FUNCTION_BLOCK FB_LidFeeder
VAR_INPUT
	_CONTROL_:BOOL;	
	bEnable:BOOL;						//Zezowlenie na pracę podajnika platynek
	bEStop:BOOL;						//Stop awaryjny nieaktywny
	bHeaterEnable:BOOL; 				//Zezwolenie na pracę grzałki wstępnej
	bRunPrepare:BOOL;							//Zezwolenie na podanie platynki. Podajnik platynek podczas cyklu podawania musi mieć załączony ten bit. Po wykonaniu podawania (kiedy status podajnika jest "LidPutted"), bit powinien być wyłączony. Dopiero kolejne załączenie pozwoli na podanie platynki
	bRun: BOOL;						//Zezwolenie na ostatni ruch opuszczania platynki
	bHoming:BOOL;						//Zezwolenie na wykonanie bazowania i pozycjonowania podajnika
	bHeightSet:BOOL;					//Ustaw wysokość
	bIgnoreError:BOOL;					//Ignorowania błędów cyklu pracy
	bReset:BOOL;						//Reset błędu, jeśli w stanie "eError"
	nLidHeatingTime:INT;				//Czas zgrzewania wstępnego [ms]
	nPositionHeightSV:LREAL;			//Wysokość zadana na której ma znajdować się podajnik
	bHeaterTemperatureErrorIgnore:BOOL; //Zmienna pozwalająca ignorowanie aktualnej temperatury
	bManualMovement:BOOL; 			//Uruchomienie trybu ruchów ręcznych
	HEATER_PARAMETERS_:BOOL;	
	nHeaterTemperatureSV:INT;			//Zadana wartość grzałki podajnika platynek
	rKp:REAL;							//Wzmocnienie proporcjonalne regulatora grzałki
	rTd:REAL;							//Czas różniczkowania regulatora grzałki
	rTi:REAL;							//Czas całkowania regulatora grzałki
	//nCycle:INT;						//Czas okresu PWM grzałki [s]
	nTempHisteresis:INT;				//Dopuszczalna różnica pomiędzy wartością zadaną a aktualną [st. C]				
	lrMaxHeight:LREAL;					//Maksymalna wysokość podajnika platynek
	lrMinHeight:LREAL;					//Minimalna wysokość podajnika platynek

	_SENSORS_:BOOL;
	bFeederActuatorUpSensor1:BOOL;		//krańcówka górna podajnika platynek
	bFeederActuatorDownSensor1:BOOL;	//krańcówka dolna podajnika platynek
	bFeederActuatorDownSensor2:BOOL;	//krańcówka dolna podajnika platynek
	bLidSuckedSensor:BOOL;				//Czujnik zassania platynki, zassana jesli TRUE
	lrHeaterTemperatureCVSensor:LREAL;	//Wartość aktualna temperatury grzałki
	bTemperatureSensorFault:BOOL;		//Błąd czujnika temperatury
	nPositionHeightCV:LREAL;			//Aktualna wysokość podajnika platynek

	_HEIGHTMOTOR_ :BOOL;	
	bHeightMotorEncoderPulse :BOOL;			//Sygnał impulsów enkodera siłownika
	rHeightMotorPositionOffset :REAL;		//Wysokość bazowani podnośnika

	_ALARMINFO_ :BOOL;
	iStationIndex:UDINT;					//Numer stacji 
	sStationName:STRING;					//Nazwa stacji	

	bLidFeederLowLevelSensor			: BOOL;		// Czujnik niskiego poziomu platynek w zasobniku
	bEmergencyUp						: BOOL;		
	//Vasyl 24.10.25 aktualizacja bloczka enkodera
	udiHeightMotorEncoderCV		: UDINT;
	bHeightEncoderSetCDone		: BOOL;	
	
END_VAR
VAR_OUTPUT
	bHeaterPWMOut :BOOL;					//Wyjscie PWM sterujące grzałką
	eState: E_Station;						//Stan ogólny bloku
	eRunningState: E_LidFeederState;		//Stan podajnika platynek
	bError: BOOL;							//Błąd stacji
	nErrorNr: UDINT;						//Nr błędu podajnika platynek
	sErrorDescription:STRING(200);			//Opis błędu
	sErrorDescription2: STRING(200);		//Opis błędu 2
	sErrorStationName:STRING;				//Nazwa stacji
	udiStationID:UDINT;						// Nr stacji

	bLidFeederActuator1:BOOL;				//Sterownie siłownika podajnika platynek
	bLidFeederActuator2:BOOL;				//Sterownie siłownika podajnika platynek
	bLidHeaterActuator:BOOL;				//Sterowanie siłownika grzałki wstępnej
	bLidSuckerActuator:BOOL;				//Sterowanie zasysaniem platynek
	bHeightMotorUp:BOOL;					//Sterowanie silnikiem podnośnika  - RUCH W GÓRĘ
	bHeightMotorDown:BOOL;					//Sterowanie silnikiem podnośnika  - RUCH W DÓŁ
	lrHeightMotorCV:LREAL;					//Aktualna pozycja podnośnika
	tCycleTime:TIME;	
	bHomingDone:BOOL;						//Wymagane ponowne bazowanie (blad podczas bazowania lub stop awaryjny)	
	bCycleDone:BOOL;
	bCycleNotDone:BOOL;
	//Vasyl 24.10.25 aktualizacja bloczka enkodera
	udiHeightMotorEncoderSetCV	: UDINT;		
	bHeightEncoderSetC			: BOOL;					// Zerowanie enkodera
	
END_VAR
VAR
	nSuckingRetry: INT;						//Licznik nieudanego pobrania platynki
	tonHeatingTime: TON;					//Timer czasu zgrzewania platynki
	tonLidSuckingDelay: TON; 				//Timer opóźnienia zassania po włączeniu eżektora w stanie zasysania
	tonHeightNoChange: TON; 				//Timer wykrycia braku ruchu siłownika zmiany wysokości stacji
	nLastPositionHeightCV: LREAL;			//Pozycja podnośnika w poprzednim cyklu programu
	tonErrorHeightChange: TON; 				//Timer błędu podnośnika

	rtEncoderHomed:R_TRIG;
	tonCycleTimer:TON;
	rtrigCycleTimerRead:R_TRIG;
	
	tonLimitPosMinReachedDelay: TON;
	tonLimitPosMaxReachedDelay: TON;
	tonMaxHeight: TON;
	tonLidFeederActuator1DownError: TON;
	tonLidFeederActuator1UpError: TON;
	tonLidFeederActuator2DownError: TON;
	//Podnośnik Jiesang	
	fbHeightMotorEncoder: FB_JiesangActuatorEncoderModul;	// Blok enkodera podnośnika chwytaka stabilizującego pod zakręcarką	
	bHeightMotorEncoderCounterReset:BOOL; 				//Sygnał resetu enkodera
	bHeightMotorEncoderHomed:BOOL;						//Informacja od enkodera że jest zbazowany

	eLastState: E_Station;							//Stan ogólny bloku
	eLastRunningState: E_LidFeederState;			//Stan podbloku
	eLastStateTemp: E_Station;						//Stan ogólny bloku
	eLastRunningStateTemp: E_LidFeederState;		//Stan podbloku
	bStateError: BOOL;
	tonEstopDelay: TON;
	
	fbTempRegulator				: FB_TempRegulator;
	bTempRegulatorReset			: BOOL;
	
	tofbHeaterPWMOut					: TOF;
	tonHeaterOnAndNotHeating			: TON;
	lrHeaterTemperatureCVSensorLast		: LREAL;	//Wartość aktualna temperatury grzałki
	tonHeaterOnAndSensorShows0			: TON;
	tofHeightMotorDown: TOF;
	tonbLidFeederLowLevelSensor: TON;
	ftWarning: F_TRIG;
	tonbLidFeederWellLevel: TON;
	rtbHeightMotorEncoderPulse: R_TRIG;
	ftbHeightMotorEncoderPulse: F_TRIG;
	lrHeightMotorEncoderPulses: LREAL;

	bLidFeederActuator1LastState		: BOOL;	//Stan przed Manual
	bLidFeederActuator2LastState		: BOOL;	//Stan przed Manual
	bLidSuckerActuatorLastState			: BOOL;	//Stan przed Manual
	bLidHeaterActuatorLastState			: BOOL;	//Stan przed Manual
	tonGoingUp: TON;
	
	//Zmienne od EVENTLOGGER
	bAlarmInit 						: BOOL := TRUE; 
	nAlarmNumerator					: INT;
	arfbAlarm						: ARRAY[0..19] OF  FB_TcAlarm;		//Tablica bloczków błędów
	fbSourceInfo 					: FB_TcSourceInfo;
	iSourceInfo						: I_TcSourceInfo;
	sAlarmTest						: STRING;
	//Koniec zmiennych od EVENTLOGGER
END_VAR

VAR_IN_OUT
	bManualLidFeederActuator1:BOOL;		//Ruch ręczny siłownikiem podajnika platynek
	bManualLidFeederActuator2:BOOL;		//Ruch ręczny siłownikiem 2 podajnika platynek
	bManualLidSuckerActuator:BOOL;		//Ręczne załączenie zassania platynek
	bManualLidHeaterActuator:BOOL;		//Ruch ręczny siłownika grzałek;
	bManualHeightMotorUp:BOOL;			//Ruch ręczny podnośnika stacji w górę
	bManualHeightMotorDown:BOOL;		//Ruch ręczny podnośnika stacji w dół
	
	bWarning							: BOOL;
END_VAR

Signals();
HeightMotor();
ErrorHandling();
Control();
HeaterRegulator();
Statistics();
EncoderTest();
aStationID();
(*Zapisywanie ostatniego stanu*)
IF eLastStateTemp<>eState THEN
	eLastState := eLastStateTemp;
END_IF
eLastStateTemp := eState;
IF eLastRunningStateTemp<>eRunningState THEN
	eLastRunningState := eLastRunningStateTemp;
END_IF
eLastRunningStateTemp := eRunningState;
(*Koniec Zapisywanie ostatniego stanu*)

nLastPositionHeightCV:=nPositionHeightCV;

ACTION aStationID:
udiStationID	:=	iStationIndex;
END_ACTION

ACTION Control:

	(** TIMERY**)
	rtEncoderHomed(CLK:=bHeightMotorEncoderHomed,Q=>);
	tonHeightNoChange(IN:=((bHeightMotorUp OR bHeightMotorDown) AND nLastPositionHeightCV=nPositionHeightCV), PT:=T#1S); 
	tonLimitPosMinReachedDelay(IN:=(nPositionHeightCV<=lrMinHeight) AND eState=E_Station.eHoming,PT:=T#2S);
	tonLimitPosMaxReachedDelay(IN:=(nPositionHeightCV>=lrMaxHeight) AND eState=E_Station.eHoming,PT:=T#2S);

	(*****Wyłączenie enable*****)
	IF NOT bEnable THEN
		IF eState <> E_Station.eDisabled AND eState <> E_Station.ePreparingToDisable THEN
				eState 				:= E_Station.ePreparingToDisable; 
		END_IF	
	END_IF

	(*****Estop*****)
	IF NOT bEstop  THEN	
		IF eState <> E_Station.eAborted AND eState <> E_Station.eAborting AND eState <> E_Station.eDisabled THEN
				eState 				:= E_Station.eAborting; 
		END_IF
	END_IF
	
	IF bEstop AND bEmergencyUp THEN
		eState 				:= E_Station.eAborting;
	END_IF

	
	CASE eState OF
	/////////////////////////////	
		E_Station.eDisabled: 					// Stan nieaktywnosci (Stacja wyłączona) 
		
			IF bEnable THEN
				eState 				:= E_Station.ePreparingToReady; 
			END_IF 
			
    /////////////////////////////	    
		E_Station.eAborted: 					// Stan bezpiecznego zatrzymania (po Abortingu) 

			IF bEStop THEN
				eState 				:= E_Station.ePreparingToReady;
			END_IF
			
	/////////////////////////////	
		E_Station.eAborting:                 	// Stan bezpiecznego zatrzymywania (po EStopie)
		
			IF NOT bEstop THEN
				
				bLidFeederActuator1		:=	FALSE;
				bLidFeederActuator2		:=	FALSE;
				bLidSuckerActuator		:=	FALSE;
				bLidHeaterActuator		:=	FALSE;
				bHeightMotorDown		:=	FALSE;
				bHeightMotorUp			:=	FALSE;	
				eState 					:=	E_Station.eAborted;  
				eRunningState			:=	E_LidFeederState.eDisabled;
				
			ELSIF bEmergencyUp THEN
			
				bHeightMotorUp			:= NOT tofHeightMotorDown.Q;
				bHeightMotorDown		:= FALSE;
				bLidFeederActuator1		:= FALSE;
				bLidFeederActuator2		:= FALSE;
				bLidSuckerActuator		:= FALSE;	
				bHeightMotorDown		:= FALSE;
				
				bHomingDone 			:= FALSE;
				
				IF tonHeightNoChange.Q THEN
					bHeightMotorEncoderCounterReset	:= TRUE;
					bHeightMotorUp					:= FALSE;
				END_IF
				
				
			END_IF
	/////////////////////////////			
		E_Station.eError:                 	 	// Stan błędu 	
		
					bLidFeederActuator1	:=FALSE;
		            bLidFeederActuator2	:=FALSE;
					bLidSuckerActuator	:=FALSE;
	
			IF bReset THEN
				eState 				:= E_Station.eResetting;
			END_IF
			
	/////////////////////////////
		E_Station.eResetting:					// Stan resetowania bledu (po Errorze)

		
// 			CASE nErrorNr-iStationIndex OF
// 		
// 				//Error 1 - ZBYT DLUGIE ZASYSANIE
// 				221:
// 					bError := FALSE;
// 				ELSE
// 					bError := FALSE;	
// 		END_CASE
			// 			
			bLidFeederActuator1	:=FALSE;
            bLidFeederActuator2	:=FALSE;
			bLidSuckerActuator	:=FALSE;
			
			IF NOT bError THEN
				nErrorNr 			:=	0;
   				sErrorDescription 	:=	'';
				bTempRegulatorReset	:=	FALSE;
				eState 				:=	E_Station.ePreparingToReady;
			ELSE
				eState 				:=	E_Station.eError;
			END_IF
        
	/////////////////////////////
		E_Station.eManualMovement:     			// Stan ruchów manualnych  
       
			ManualMovements();
			//Wyjście z trybu serwisowego
			IF NOT bManualMovement THEN
				bLidFeederActuator1		:=	bLidFeederActuator1LastState ;//:=FALSE;
				bLidFeederActuator2		:=	bLidFeederActuator2LastState ; //:=FALSE;
				bLidSuckerActuator		:=	bLidSuckerActuatorLastState ;//:=FALSE;
				bLidHeaterActuator		:=	bLidHeaterActuatorLastState ;//:=FALSE;
				bHeightMotorDown		:=	FALSE;
				bHeightMotorUp			:=	FALSE;
				eState:=E_Station.eReady;
			END_IF

	/////////////////////////////
		E_Station.eHoming:						// Stan bazowania 

			Homing();
			IF NOT bHoming AND NOT bHeightSet THEN
			   eState:=E_Station.ePreparingToReady;
			   	bHeightMotorDown:=FALSE;
				bHeightMotorUp:=FALSE;
			END_IF		
			
	/////////////////////////////
		E_Station.eHomingDone:                  // Stan wykonania bazowania 
		
			bHeightMotorDown:=FALSE;
			bHeightMotorUp:=FALSE;
			bHeightMotorEncoderCounterReset:=FALSE;
			bHomingDone:=TRUE;
			IF NOT bHoming AND NOT bHeightSet THEN
			  	 eState:=E_Station.eReady;
			END_IF
			
	/////////////////////////////
		E_Station.ePreparingToReady:            // Stan przygotowywania do gotowosci (zawsze przed Ready)  
		
			bLidFeederActuator1		:=	FALSE;
			bLidFeederActuator2		:=	FALSE;
			//bLidSuckerActuator		:=	FALSE; //Zmiana LU205
			bLidHeaterActuator		:=	FALSE;
			eRunningState:=E_LidFeederState.eReady;
			eState:=E_Station.eReady;	
			
	/////////////////////////////
		E_Station.ePreparingToDisable:          // Stan przygotowywania do nieaktywnosci (po wyłączeniu Enable) 
  
			bLidFeederActuator1		:=	FALSE;
			bLidFeederActuator2		:=	FALSE;
			bLidSuckerActuator		:=	FALSE;
			bLidHeaterActuator		:=	FALSE;
			
			bHeightMotorUp:=TRUE;
			bHeightMotorDown:=FALSE;	
			IF tonHeightNoChange.Q THEN
				bHeightMotorUp:=FALSE;
				bHeightMotorDown:=FALSE;	
				eState:=E_Station.eDisabled;
				eRunningState:=E_LidFeederState.eDisabled;
			END_IF
			
			
	/////////////////////////////
		E_Station.eReady:						// Stan gotowosci 
		
			IF bRunPrepare OR bRun AND (NOT bCycleDone AND NOT bCycleNotDone) THEN
				eState 				:= E_Station.eStarting; 
			END_IF
			IF bHoming OR bHeightSet THEN
				eState 				:= E_Station.eHoming; 
			END_IF
			IF bManualMovement THEN
				//Jeśli przejście w tryb ruchów manualnych przepisz wszystkie stany siłowników sterowanych przez moduł
				//aby zapobiec ewentualnym kolizjom po wejściu w tryb serwisowy
				bManualLidFeederActuator1	:= bLidFeederActuator1LastState :=	bLidFeederActuator1;
				bManualLidFeederActuator2	:= bLidFeederActuator2LastState :=	bLidFeederActuator2;
				bManualLidSuckerActuator	:= bLidSuckerActuatorLastState 	:=  bLidSuckerActuator;
				bManualLidHeaterActuator	:= bLidHeaterActuatorLastState	:=	bLidHeaterActuator;
				bManualHeightMotorUp		:=	bHeightMotorUp;
				bManualHeightMotorDown		:=	bHeightMotorDown;
				
				eState 						:=	E_Station.eManualMovement; 
			END_IF
			IF NOT bRun THEN
				bCycleDone 					:= FALSE;
				bCycleNotDone 				:= FALSE;			
			END_IF
			
	/////////////////////////////
		E_Station.eStopping:					// Stan zatrzymywania 
		
			Running();
			IF eRunningState=E_LidFeederState.eReady THEN
				eState 	:= E_Station.eReady;
			END_IF
			//eState 					:= E_Station.eReady;	
			
	/////////////////////////////
		E_Station.eStarting:                  	// Stan uruchamiania (po Ready)
		
			eState					 := E_Station.eRunning; 
			
	/////////////////////////////
		E_Station.eRunning:              		// Stan wykonywania cyklu (po Startingu), w tym stanie osobny
 
			Running();
			IF NOT bRunPrepare THEN					(*Przerywanie cyklu*)
				eState 				 := E_Station.eStopping;	
			END_IF
			IF bCycleDone OR bCycleNotDone THEN (*Cykl zakończony*)
				eState 				 := E_Station.eReady;
			END_IF	
	/////////////////////////////		
	END_CASE
END_ACTION

ACTION EncoderTest:


rtbHeightMotorEncoderPulse(CLK:=bHeightMotorEncoderPulse,Q=>);
ftbHeightMotorEncoderPulse(CLK:=bHeightMotorEncoderPulse,Q=>);


IF rtbHeightMotorEncoderPulse.Q THEN
	lrHeightMotorEncoderPulses	:=	lrHeightMotorEncoderPulses +	1;
END_IF
END_ACTION

ACTION ErrorHandling:
// Alarm_0340	340	Error	Zbyt długa próba zassania platynki - uzupełnij platynki lub popraw ich położenie
// Alarm_0341	341	Error	Nieudana próba podania platynki - zwiększ ciśnienie
// Alarm_0342	342	Error	Błąd czujnika temperatury grzałki - sprawdź połączenie
// Alarm_0343	343	Error	Blokada podnośnika lub brak zasilania - sprawdź czujnik lub odblokuj mechanicznie
// Alarm_0344	344	Error	Wartość zadana wysokości jest większa od maksymalnej - zmień ustawienia w recepturze
// Alarm_0345	345	Error	Blokada siłownika dolnego podczas opuszczania - sprawdź czujnik
// Alarm_0346	346	Error	Blokada siłownika dolnego podczas podnoszenia - sprawdź czujnik
// Alarm_0347	347	Error	Blokada siłownika górnego podczas opuszczania - sprawdź czujnik
// Alarm_0348	348	Error	Błąd grzania, brak wzrostu temperatury - sprawdź czujnik
// Alarm_0349	349	Error	Błąd grzania, brak sygnału z czujnika temperatury - sprawdź czujnik

IF bAlarmInit THEN
    bAlarmInit := FALSE; 
	fbSourceInfo.Clear();
	fbSourceInfo.sName:=sStationName;//'Machine';
	fbSourceInfo.nId:=udiStationID;//2700;
	// Alarm_0340	340	Error	Zbyt długa próba zassania platynki - uzupełnij platynki lub popraw ich położenie
    arfbAlarm[0].CreateEx(stEventEntry := TC_EVENTS.AlarmClass.Alarm_0340, bWithConfirmation:= FALSE,  ipSourceInfo:= fbSourceInfo); 
	// Alarm_0341	341	Error	Nieudana próba podania platynki - zwiększ ciśnienie
	arfbAlarm[1].CreateEx(stEventEntry := TC_EVENTS.AlarmClass.Alarm_0341, bWithConfirmation:= FALSE,  ipSourceInfo:= fbSourceInfo); 
	//// Alarm_0342	342	Error	Błąd czujnika temperatury grzałki - sprawdź połączenie
	//arfbAlarm[2].CreateEx(stEventEntry := TC_EVENTS.AlarmClass.Alarm_0342, bWithConfirmation:= FALSE,  ipSourceInfo:= fbSourceInfo); 
	// Alarm_0343	343	Error	Blokada podnośnika lub brak zasilania - sprawdź czujnik lub odblokuj mechanicznie
	arfbAlarm[3].CreateEx(stEventEntry := TC_EVENTS.AlarmClass.Alarm_0343, bWithConfirmation:= FALSE,  ipSourceInfo:= fbSourceInfo); 
	// Alarm_0344	344	Error	Wartość zadana wysokości jest większa od maksymalnej - zmień ustawienia w recepturze
	arfbAlarm[4].CreateEx(stEventEntry := TC_EVENTS.AlarmClass.Alarm_0344, bWithConfirmation:= FALSE,  ipSourceInfo:= fbSourceInfo); 
	// Alarm_0345	345	Error	Blokada siłownika dolnego podczas opuszczania - sprawdź czujnik
	arfbAlarm[5].CreateEx(stEventEntry := TC_EVENTS.AlarmClass.Alarm_0345, bWithConfirmation:= FALSE,  ipSourceInfo:= fbSourceInfo); 
	// Alarm_0346	346	Error	Blokada siłownika dolnego podczas podnoszenia - sprawdź czujnik
	arfbAlarm[6].CreateEx(stEventEntry := TC_EVENTS.AlarmClass.Alarm_0346, bWithConfirmation:= FALSE,  ipSourceInfo:= fbSourceInfo); 
	// Alarm_0347	347	Error	Blokada siłownika górnego podczas opuszczania - sprawdź czujnik
	arfbAlarm[7].CreateEx(stEventEntry := TC_EVENTS.AlarmClass.Alarm_0347, bWithConfirmation:= FALSE,  ipSourceInfo:= fbSourceInfo); 
	//// Alarm_0348	348	Error	Błąd grzania, brak wzrostu temperatury - sprawdź czujnik
	//arfbAlarm[8].CreateEx(stEventEntry := TC_EVENTS.AlarmClass.Alarm_0348, bWithConfirmation:= FALSE,  ipSourceInfo:= fbSourceInfo); 
	//// Alarm_0349	349	Error	Błąd grzania, brak sygnału z czujnika temperatury - sprawdź czujnik
	//arfbAlarm[9].CreateEx(stEventEntry := TC_EVENTS.AlarmClass.Alarm_0349, bWithConfirmation:= FALSE,  ipSourceInfo:= fbSourceInfo); 
END_IF



//OBSŁUGA BŁĘDÓW 


////GRZAŁKI NIEGOTOWE (różnica temperatury grzałki różna od zadanej +/-10 st.C 
//IF (ABS(lrHeaterTemperatureCVSensor-nHeaterTemperatureSV)>nTempHisteresis AND bHeaterEnable AND NOT bHeaterTemperatureErrorIgnore) AND eState=E_Station.eReady AND NOT bHoming THEN
//		eRunningState:=E_LidFeederState.eHeaterNotReady;	
//ELSIF eRunningState=E_LidFeederState.eHeaterNotReady THEN																							//zmiana 11
//		IF (ABS(lrHeaterTemperatureCVSensor-nHeaterTemperatureSV)<nTempHisteresis OR bHeaterTemperatureErrorIgnore) OR NOT bHeaterEnable OR bHoming THEN
//			eRunningState:=E_LidFeederState.eReady;	
//		END_IF	
//END_IF
//tonEstopDelay			(IN:=bEstop,	PT:=T#5S); //Opóżnienie po EStopie w celu blokoady błędów, powietrze jest później niż Estop a sygnał z czujnika nie pokazuje braku powietrza bo jest odcinany za tym


//************LISTA BŁĘDÓW***************
bStateError:= (eState=E_Station.eError) OR (eState=E_Station.eResetting);(* OR bIgnoreError; *)

IF bEnable THEN
	// Alarm_0340	340	Error	Zbyt długa próba zassania platynki - uzupełnij platynki lub popraw ich położenie
	//Error 1 - ZA DŁUGA PRÓBA ZASYSANIA PLATYNKI
	tonLidSuckingDelay(IN:=(eRunningState=E_LidFeederState.eSuckingLid AND NOT bLidSuckedSensor),PT:=T#1S);
	IF tonLidSuckingDelay.Q AND NOT bStateError THEN
		IF NOT arfbAlarm[0].bActive THEN
			bLidSuckerActuator:=FALSE;
			arfbAlarm[0].Raise(nTimeStamp:=0);
		END_IF
	ELSE	
		IF  arfbAlarm[0].bActive AND bReset THEN
			arfbAlarm[0].Clear(nTimeStamp:=0, bResetConfirmation:= FALSE);
		END_IF	
//		bLidSuckerActuator:=FALSE;
// 		bError := TRUE;
// 		nErrorNr:=221;
// 		//nErrorNr := nErrorNr+iStationIndex;
// 		sErrorDescription:='Zbyt długa próba zassania platynki - uzupełnij platynki lub popraw ich położenie';
// 		eRunningState:=E_LidFeederState.eReady;
	END_IF;
	// Alarm_0341	341	Error	Nieudana próba podania platynki - zwiększ ciśnienie
	//Error 2 - TRZYKROTNE ODERWANIE SIĘ PLATYNKI PRZY PRÓBIE PODANIA
	IF (nSuckingRetry>=3) THEN
		IF NOT arfbAlarm[0].bActive THEN
			nSuckingRetry:=0;
			bLidSuckerActuator:=FALSE;
			bLidFeederActuator1:=FALSE;
			arfbAlarm[0].Raise(nTimeStamp:=0);
		END_IF
	ELSE	
		IF  arfbAlarm[0].bActive AND bReset THEN
			arfbAlarm[0].Clear(nTimeStamp:=0, bResetConfirmation:= FALSE);
		END_IF	
// 		nSuckingRetry:=0;
// 		bLidSuckerActuator:=FALSE;
// 		bLidFeederActuator1:=FALSE;
// 		bError := TRUE;
// 		nErrorNr:=222;
// 		//nErrorNr := nErrorNr+iStationIndex;
// 		sErrorDescription:='Nieudana próba podania platynki - zwiększ ciśnienie';
	END_IF;
//	// Alarm_0342	342	Error	Błąd czujnika temperatury grzałki - sprawdź połączenie
//	//Error 3 - Błąd czujnika temperatury
//	IF bHeaterEnable AND bTemperatureSensorFault THEN
//		IF NOT arfbAlarm[2].bActive THEN
//			bTempRegulatorReset:=TRUE;	
//			arfbAlarm[2].Raise(nTimeStamp:=0);
//		END_IF
//	ELSE	
//		IF  arfbAlarm[2].bActive AND bReset THEN
//			arfbAlarm[2].Clear(nTimeStamp:=0, bResetConfirmation:= FALSE);
//		END_IF	
//// 		bTempRegulatorReset:=TRUE;	
//// 		bError := TRUE;
//// 		nErrorNr:=223;
//// 		//nErrorNr := nErrorNr+iStationIndex;
//// 		sErrorDescription:='Błąd czujnika temperatury grzałki - sprawdź połączenie';
//	END_IF;
	// Alarm_0343	343	Error	Blokada podnośnika lub brak zasilania - sprawdź czujnik lub odblokuj mechanicznie
	//Error 4 - podnośnik nie porusza się pomimo wysterowania 
	tonErrorHeightChange(IN:=(bHeightMotorUp OR bHeightMotorDown) AND nLastPositionHeightCV=nPositionHeightCV, PT:=T#3S);
	IF tonErrorHeightChange.Q THEN
		IF NOT arfbAlarm[3].bActive THEN
			bHeightMotorUp:=FALSE;
			bHeightMotorDown:=FALSE;
			arfbAlarm[3].Raise(nTimeStamp:=0);
		END_IF
	ELSE	
		IF  arfbAlarm[3].bActive AND bReset THEN
			arfbAlarm[3].Clear(nTimeStamp:=0, bResetConfirmation:= FALSE);
		END_IF
// 		bHeightMotorUp:=FALSE;
// 		bHeightMotorDown:=FALSE;
// 		bError := TRUE;
// 		nErrorNr:=224;
// 		//nErrorNr := nErrorNr+iStationIndex;
// 		sErrorDescription:='Blokada podnośnika lub brak zasilania - sprawdź czujnik lub odblokuj mechanicznie';	
	END_IF
	// Alarm_0344	344	Error	Wartość zadana wysokości jest większa od maksymalnej - zmień ustawienia w recepturze
	//Error 5 - Bład nastaw max
	tonMaxHeight(IN:=nPositionHeightSV>lrMaxHeight AND NOT bHomingDone AND eState=E_Station.eReady,PT:=T#30S);
	IF tonMaxHeight.Q THEN
		arfbAlarm[4].ipArguments.Clear() .AddLReal(lrMaxHeight);
		IF NOT arfbAlarm[4].bActive THEN
			bHeightMotorUp:=FALSE;
			bHeightMotorDown:=FALSE;
			arfbAlarm[4].Raise(nTimeStamp:=0);
		END_IF
	ELSE	
		IF  arfbAlarm[4].bActive AND bReset THEN
			arfbAlarm[4].Clear(nTimeStamp:=0, bResetConfirmation:= FALSE);
		END_IF
// 		bHeightMotorUp:=FALSE;
// 		bHeightMotorDown:=FALSE;
// 		bError := TRUE;
// 		nErrorNr:=225;
// 		//nErrorNr := nErrorNr+iStationIndex;
// 		sErrorDescription:='Wartość zadana wysokości jest większa od maksymalnej - zmień ustawienia w recepturze';
// 		sErrorDescription2:=REAL_TO_STRING(LREAL_TO_INT(lrMaxHeight));
	END_IF
	// Alarm_0345	345	Error	Blokada siłownika dolnego podczas opuszczania - sprawdź czujnik
	//Error 6 - Zacięcie siłownika 1 odkładania platynki	
	tonLidFeederActuator1DownError(IN:=(bLidFeederActuator1 AND NOT bFeederActuatorDownSensor1 AND NOT bLidFeederActuator2),PT:= T#4S(*T#2S*)); //Add NOT bLidFeederActuator2 26.04.2023
	IF tonLidFeederActuator1DownError.Q THEN
		IF NOT arfbAlarm[5].bActive THEN
			bLidFeederActuator1:=FALSE;
			bLidFeederActuator2:=FALSE;		
			arfbAlarm[5].Raise(nTimeStamp:=0);
		END_IF
	ELSE	
		IF  arfbAlarm[5].bActive AND bReset THEN
			arfbAlarm[5].Clear(nTimeStamp:=0, bResetConfirmation:= FALSE);
		END_IF
// 		//bLidSuckerActuator:=FALSE;
// 		bLidFeederActuator1:=FALSE;
// 		bLidFeederActuator2:=FALSE;		
// 		bError := TRUE;
// 		nErrorNr:=226;
// 		//nErrorNr := nErrorNr+iStationIndex;
// 		sErrorDescription:='Blokada siłownika dolnego podczas opuszczania - sprawdź czujnik';	
	END_IF;
	// Alarm_0346	346	Error	Blokada siłownika dolnego podczas podnoszenia - sprawdź czujnik
	//Error 7 - Zacięcie siłownika 1 odkładania platynki	
	tonLidFeederActuator1UpError(IN:=NOT bLidFeederActuator1 AND NOT bFeederActuatorUpSensor1 AND tonEstopDelay.Q,PT:=(*T#2S*)T#4S);
	IF tonLidFeederActuator1UpError.Q THEN
		IF NOT arfbAlarm[6].bActive THEN
			bLidFeederActuator1:=FALSE;
			bLidFeederActuator2:=FALSE;	
			arfbAlarm[6].Raise(nTimeStamp:=0);
		END_IF
	ELSE	
		IF  arfbAlarm[6].bActive AND bReset THEN
			arfbAlarm[6].Clear(nTimeStamp:=0, bResetConfirmation:= FALSE);
		END_IF
		//bLidSuckerActuator:=FALSE; //Zmiana LU205
// 		bLidFeederActuator1:=FALSE;
// 		bLidFeederActuator2:=FALSE;		
// 		bError := TRUE;
// 		nErrorNr:=227;
// 		//nErrorNr := nErrorNr+iStationIndex;
// 		sErrorDescription:='Blokada siłownika dolnego podczas podnoszenia - sprawdź czujnik';	
	END_IF;	
	// Alarm_0347	347	Error	Blokada siłownika górnego podczas opuszczania - sprawdź czujnik
	//Error 8 - Zacięcie siłownika 2 odkładania platynki	
	tonLidFeederActuator2DownError(IN:=bLidFeederActuator2 AND NOT bFeederActuatorDownSensor2,PT:=T#2S);
	IF tonLidFeederActuator2DownError.Q THEN
		IF NOT arfbAlarm[7].bActive THEN
			bLidSuckerActuator:=FALSE;
			bLidFeederActuator1:=FALSE;
			bLidFeederActuator2:=FALSE;	
			arfbAlarm[7].Raise(nTimeStamp:=0);
		END_IF
	ELSE	
		IF  arfbAlarm[7].bActive AND bReset THEN
			arfbAlarm[7].Clear(nTimeStamp:=0, bResetConfirmation:= FALSE);
		END_IF
// 		bLidSuckerActuator:=FALSE;
// 		bLidFeederActuator1:=FALSE;
// 		bLidFeederActuator2:=FALSE;		
// 		bError := TRUE;
// 		nErrorNr:=228;
// 		//nErrorNr := nErrorNr+iStationIndex;
// 		sErrorDescription:='Blokada siłownika górnego podczas opuszczania - sprawdź czujnik';	
	END_IF;		
//	// Alarm_0348	348	Error	Błąd grzania, brak wzrostu temperatury - sprawdź czujnik
//	//Error 9 - Błąd czujnika temperatury
//	tofbHeaterPWMOut(IN:=bHeaterPWMOut,PT:=T#30S);
//	tonHeaterOnAndNotHeating(IN:=tofbHeaterPWMOut.Q AND lrHeaterTemperatureCVSensor=lrHeaterTemperatureCVSensorLast AND NOT bIgnoreError , PT:=T#5M);
//	lrHeaterTemperatureCVSensorLast := lrHeaterTemperatureCVSensor;
//	IF tonHeaterOnAndNotHeating.Q THEN
//		IF NOT arfbAlarm[8].bActive THEN
//			bTempRegulatorReset 	:= TRUE;
//			arfbAlarm[8].Raise(nTimeStamp:=0);
//		END_IF
//	ELSE	
//		IF  arfbAlarm[8].bActive AND bReset THEN
//			arfbAlarm[8].Clear(nTimeStamp:=0, bResetConfirmation:= FALSE);
// 		END_IF	
////  		bTempRegulatorReset 	:= TRUE;
//// 		bError 					:= TRUE;
//// 		nErrorNr 				:= 229;
//// 		//nErrorNr				:=nErrorNr+iStationIndex;
//// 		sErrorDescription 		:= 'Błąd grzania, brak wzrostu temperatury - sprawdź czujnik';	
//	END_IF
//	// Alarm_0349	349	Error	Błąd grzania, brak sygnału z czujnika temperatury - sprawdź czujnik
//	//Error 10 - Błąd czujnika temperatury, wskazuje 0
//	tonHeaterOnAndSensorShows0(IN:=bHeaterPWMOut AND lrHeaterTemperatureCVSensor<1 AND NOT bIgnoreError , PT:=T#15S);
//	IF tonHeaterOnAndSensorShows0.Q THEN
//		IF NOT arfbAlarm[9].bActive THEN
//			bTempRegulatorReset 	:= TRUE;
//			arfbAlarm[9].Raise(nTimeStamp:=0);
//		END_IF
//	ELSE	
//		IF  arfbAlarm[9].bActive AND bReset THEN
//			arfbAlarm[9].Clear(nTimeStamp:=0, bResetConfirmation:= FALSE);
// 		END_IF	
////  		bTempRegulatorReset 	:= TRUE;
//// 		bError 					:= TRUE;
//// 		nErrorNr 				:= 230;
//// 		//nErrorNr				:=nErrorNr+iStationIndex;
//// 		sErrorDescription 		:= 'Błąd grzania, brak sygnału z czujnika temperatury - sprawdź czujnik';	
//	END_IF
	
// Warning czujnik poziomu	
	tonbLidFeederLowLevelSensor( IN:= bLidFeederLowLevelSensor, PT:= T#10S);
	
	IF tonbLidFeederLowLevelSensor.Q THEN
		bWarning				:= TRUE;
	END_IF
	
	tonbLidFeederWellLevel( IN:= bLidFeederLowLevelSensor, PT:= T#1S);	
	
	IF tonbLidFeederWellLevel.Q THEN
		bWarning				:= FALSE;
	END_IF	
	
	ftWarning(CLK:=bWarning);
	
	IF ftWarning.Q THEN
		tonbLidFeederLowLevelSensor( IN:= FALSE);
	END_IF
	
	
ELSE
		bError 					:= FALSE;
END_IF
//*******KONIEC LISTA BŁĘDÓW***************


//******************PRZEJŚCIE DO eERROR*****************************

IF bError AND NOT bStateError THEN
	IF eLastState = eRunning THEN
		bCycleNotDone := TRUE;
	END_IF
	eState := E_Station.eError;
END_IF

//****************WYŚWIETLANIE STATUSU BLEDU***********************


(*Wyświetlanie błedu na wyjściu*)
bError							:= FALSE;
FOR nAlarmNumerator := 0 TO 19 DO
	bError						:= bError OR arfbAlarm[nAlarmNumerator].bActive;
END_FOR

(*Przepisywanie nazwy stacji*)
sErrorStationName:=sStationName;



//Jezeli nie zbazowane to potrzebne bazowanie
IF NOT bHeightMotorEncoderHomed  THEN
	bHomingDone:=FALSE;
END_IF
END_ACTION

ACTION HeaterRegulator:
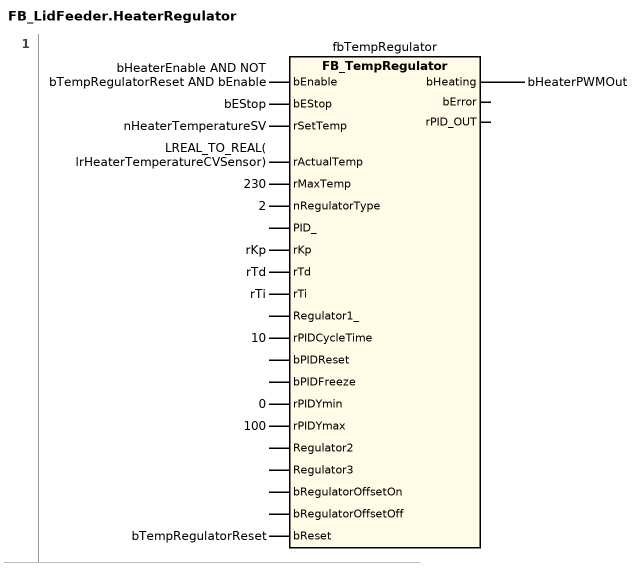
// NETWORK 1
fbTempRegulator(
    bEnable := bHeaterEnable AND NOT bTempRegulatorReset AND bEnable,
    bEStop := bEStop,
    rSetTemp := nHeaterTemperatureSV,
    rActualTemp := LREAL_TO_REAL(lrHeaterTemperatureCVSensor),
    rMaxTemp := 230,
    nRegulatorType := 2,
    rKp := rKp,
    rTd := rTd,
    rTi := rTi,
    rPIDCycleTime := 10,
    rPIDYmin := 0,
    rPIDYmax := 100,
    bReset := bTempRegulatorReset); // FB_TempRegulator
bHeaterPWMOut := fbTempRegulator.bHeating;
END_ACTION

ACTION HeightMotor:
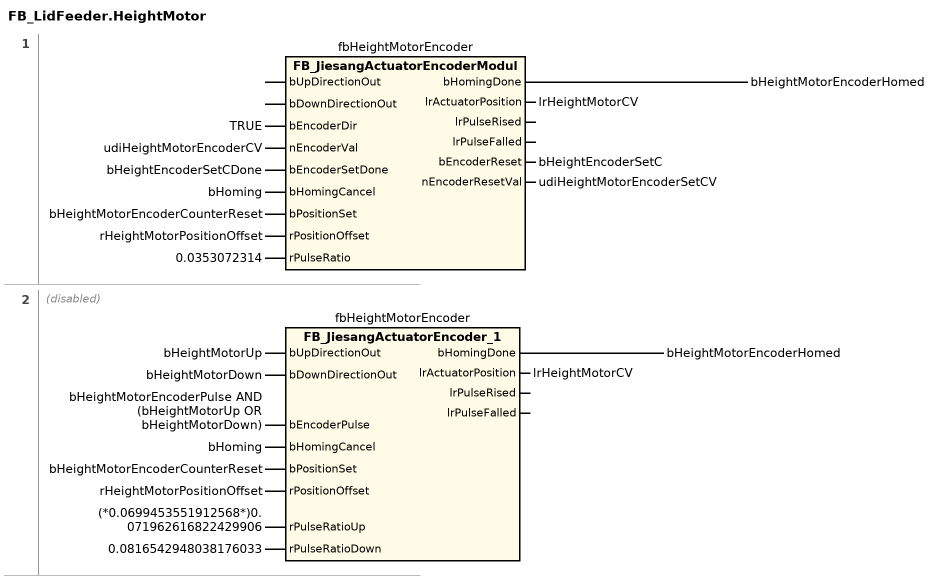
// NETWORK 1
fbHeightMotorEncoder(
    bEncoderDir := TRUE,
    nEncoderVal := udiHeightMotorEncoderCV,
    bEncoderSetDone := bHeightEncoderSetCDone,
    bHomingCancel := bHoming,
    bPositionSet := bHeightMotorEncoderCounterReset,
    rPositionOffset := rHeightMotorPositionOffset,
    rPulseRatio := 0.0353072314,
    lrActuatorPosition => lrHeightMotorCV,
    bEncoderReset => bHeightEncoderSetC,
    nEncoderResetVal => udiHeightMotorEncoderSetCV); // FB_JiesangActuatorEncoderModul
bHeightMotorEncoderHomed := fbHeightMotorEncoder.bHomingDone;

// NETWORK 2 (disabled)
// fbHeightMotorEncoder(
//     bUpDirectionOut := bHeightMotorUp,
//     bDownDirectionOut := bHeightMotorDown,
//     bEncoderPulse := bHeightMotorEncoderPulse AND (bHeightMotorUp OR bHeightMotorDown),
//     bHomingCancel := bHoming,
//     bPositionSet := bHeightMotorEncoderCounterReset,
//     rPositionOffset := rHeightMotorPositionOffset,
//     rPulseRatioUp := (*0.0699453551912568*)0.071962616822429906,
//     rPulseRatioDown := 0.0816542948038176033,
//     lrActuatorPosition => lrHeightMotorCV); // FB_JiesangActuatorEncoder_1
// bHeightMotorEncoderHomed := fbHeightMotorEncoder.bHomingDone;
END_ACTION

ACTION Homing:
//BAZOWANIE PODAJNIKA PLATYNEK

bLidFeederActuator1:=FALSE;
bLidHeaterActuator:=FALSE;
bLidSuckerActuator:=FALSE;

tofHeightMotorDown(IN:=bHeightMotorDown, PT:=T#1S); //Zabezpieczenie przed zbyt szybkim przełączeniem pomiędzy Down a Up, bezpiecznieki sie palą
	
//Podnoszenie stacji do maksymalnej pozycji
IF NOT bHeightMotorEncoderHomed OR rtEncoderHomed.Q THEN
	bHeightMotorUp		:=	(*TRUE*) NOT tofHeightMotorDown.Q;
	bHeightMotorDown	:=	FALSE;
	IF tonHeightNoChange.Q THEN
		bHeightMotorEncoderCounterReset:=TRUE;
		bHeightMotorUp:=FALSE;
	END_IF
	//Jesli enkoder zbazowany zakończ bazowanie	
	IF rtEncoderHomed.Q THEN
		bHeightMotorUp:=FALSE;
		bHeightMotorDown:=FALSE;
		eState:=E_Station.eHomingDone;
	END_IF	
//Po podniesieniu stacji opuszczanie do ustalonej wysokości
ELSIF bHeightMotorEncoderHomed THEN
	bHeightMotorEncoderCounterReset:=FALSE;
	bHeightMotorUp:=nPositionHeightCV<=nPositionHeightSV AND (nPositionHeightCV<=lrMaxHeight);
	bHeightMotorDown:=nPositionHeightCV>=nPositionHeightSV AND (nPositionHeightCV>=lrMinHeight);
	//Kiedy stacja osiągnie wysokość zadaną
	IF ABS(nPositionHeightCV-nPositionHeightSV)<1 OR tonLimitPosMinReachedDelay.Q OR tonLimitPosMaxReachedDelay.Q THEN
			bHeightMotorDown:=FALSE;
			bHeightMotorUp:=FALSE;
			eState:=E_Station.eHomingDone;
	END_IF			
END_IF
END_ACTION

ACTION ManualMovements:
//W trybie ruchów manualnych wykonuj ruchy za pomocą rozkazów manualnych
IF NOT bRunPrepare AND NOT bRun THEN
	bLidFeederActuator1:=bManualLidFeederActuator1;
	bLidFeederActuator2:=bManualLidFeederActuator2;	
	bLidSuckerActuator:=bManualLidSuckerActuator;
	bLidHeaterActuator:=bManualLidHeaterActuator ;
	bHeightMotorUp:=bManualHeightMotorUp;
	bHeightMotorDown:=bManualHeightMotorDown;
ELSE
	bManualLidFeederActuator1:=FALSE;
	bManualLidFeederActuator2:=FALSE;
	bManualLidSuckerActuator:=FALSE;
	bManualLidHeaterActuator:=FALSE;
	bManualHeightMotorUp:=FALSE;
	bManualHeightMotorDown:=FALSE;
END_IF
	
IF bHoming OR bHeightSet THEN
	eState:=E_Station.eHoming;
END_IF
	
Running();
	
//Zabezpieczenie przed kolizją stacji poprzez ruch podnośnika	
IF bHeightMotorDown AND nPositionHeightCV<=lrMinHeight AND NOT bHoming AND NOT bHeightSet THEN
	bHeightMotorDown:=FALSE;
END_IF	

IF bHeightMotorUp AND nPositionHeightCV>=lrMaxHeight AND NOT bHoming AND NOT bHeightSet THEN
	bHeightMotorUp:=FALSE;
END_IF		 		 

IF NOT bRun THEN
	bCycleDone 					:= FALSE;
	bCycleNotDone 				:= FALSE;	
END_IF
END_ACTION

ACTION Running:

//Timery 
tonHeatingTime(IN:=eRunningState=E_LidFeederState.eHeating,PT:=INT_TO_TIME(nLidHeatingTime));

CASE eRunningState OF
	
	//PODAJNIK GOTOWY DO PRACY
	E_LidFeederState.eDisabled:
			eRunningState:=E_LidFeederState.eReady;
	
	//PODAJNIK GOTOWY DO PRACY
	E_LidFeederState.eReady:
		//Jeśli komenda podania platynki przejdź do stanu zasysania platynki
		IF NOT bCycleDone AND NOT bCycleNotDone THEN	
			IF bRunPrepare OR bRun THEN
				IF bLidSuckedSensor THEN //24.04.2023 MP
					eRunningState:=E_LidFeederState.ePuttingLid;
				ELSE
					eRunningState:=E_LidFeederState.eSuckingLid;
				END_IF
				//eRunningState:=E_LidFeederState.eSuckingLid;
			END_IF
		END_IF
	
	//PODAJNIK ZASYSA PLATYNKĘ
	E_LidFeederState.eSuckingLid:
		bLidFeederActuator1:=FALSE;
		bLidFeederActuator2:=FALSE;
		bLidSuckerActuator:= bFeederActuatorUpSensor1 AND NOT bLidFeederActuator1;
		//Jeśli komenda podania platynki przejdź do stanu opuszczania siłownika podajnika
		IF bLidSuckedSensor OR bIgnoreError THEN
			eRunningState:=E_LidFeederState.ePuttingLid;
		END_IF

	//PODAJNIK OPUSZCZA PLATYNKĘ
	E_LidFeederState.ePuttingLid:
		bLidFeederActuator1:=TRUE;
		//Jeśli platynka podczas ruchu siłownika podajnika odpadnie przejdź do stanu zasysania platynki i zwiększ licznik nieudanego zassania o 1
		IF NOT (bLidSuckedSensor OR bIgnoreError ) THEN
			nSuckingRetry:=nSuckingRetry+1;
			eRunningState:=E_LidFeederState.eSuckingLid;
		END_IF
		//Jeśli platynka podczas ruchu siłownika podajnika odpadnie przejdź do stanu zasysania platynki i zwiększ licznik nieudanego zassania o 1
		IF (bLidSuckedSensor OR bIgnoreError ) AND bFeederActuatorDownSensor1 AND bRun THEN
			eRunningState:=E_LidFeederState.ePuttingLid2;
		END_IF
		
		IF NOT bRunPrepare AND NOT bRun THEN //24.04.2023 MP
			eRunningState := E_LidFeederState.eGoingUp;
			//eRunningState := E_LidFeederState.eReady;
		END_IF
	
	//PODAJNIK OPUSZCZA PLATYNKĘ CZ.2
	E_LidFeederState.ePuttingLid2:
		bLidFeederActuator2:=TRUE;
		//Jeśli platynka podczas ruchu siłownika podajnika odpadnie przejdź do stanu zasysania platynki i zwiększ licznik nieudanego zassania o 1
		IF NOT (bLidSuckedSensor OR bIgnoreError ) THEN
			nSuckingRetry:=nSuckingRetry+1;
			eRunningState:=E_LidFeederState.eSuckingLid;
		END_IF
		//Jeśli platynka zassana i siłownik osiągnął dolny poziom przejdź do stanu zgrzewania wstępnego 
		IF (bLidSuckedSensor OR bIgnoreError) AND bFeederActuatorDownSensor2 THEN
			eRunningState:=E_LidFeederState.eHeating;
			bLidSuckerActuator:=FALSE;
		END_IF		

	//PODAJNIK WSTĘPNIE ZGRZEWA PLATYNKĘ
	E_LidFeederState.eHeating:

		bLidSuckerActuator:=FALSE;
		//Zgrzewanie platynki dopóki nie osiągnie czasu przygrzewania
		IF NOT tonHeatingTime.Q THEN
			bLidFeederActuator1:=TRUE;
			bLidFeederActuator2:=TRUE;
			bLidHeaterActuator:=TRUE;
		ELSE
			bLidFeederActuator1:=FALSE;
			bLidFeederActuator2:=FALSE;
			bLidHeaterActuator:=FALSE;
			IF NOT bFeederActuatorDownSensor1 THEN
				eRunningState:=E_LidFeederState.eLidPutted;	
			END_IF
		END_IF

	//PODAJNIK WYKONAŁ ODKŁADANIE PLATYNEK
	E_LidFeederState.eLidPutted:
		bLidFeederActuator1:=FALSE;
		bLidFeederActuator2:=FALSE;
		bLidHeaterActuator:=FALSE;
		bLidSuckerActuator:=FALSE;
		nSuckingRetry:=0;
		bCycleDone := TRUE;
		IF bFeederActuatorUpSensor1 AND NOT bFeederActuatorDownSensor2 THEN
			eRunningState:=E_LidFeederState.eReady;
		ELSE
			eRunningState:=E_LidFeederState.eGoingUp;
		END_IF
	
	
	//PODAJNIK PODNOSI SIŁOWNIK PODAWANIA PLATYNEK
	E_LidFeederState.eGoingUp:
		bLidFeederActuator1:=FALSE;
		bLidFeederActuator2:=FALSE;
		bLidHeaterActuator:=FALSE;
		//bLidSuckerActuator:=FALSE;
		IF bLidSuckerActuator THEN
			IF tonGoingUp.Q AND bFeederActuatorUpSensor1 THEN
				eRunningState		:=	E_LidFeederState.eReady;
				bLidSuckerActuator	:=	FALSE;			
			END_IF
		ELSE
			IF bFeederActuatorUpSensor1 THEN
				eRunningState		:=	E_LidFeederState.eReady;
				bLidSuckerActuator	:=	FALSE;
			END_IF
		END_IF


END_CASE
END_ACTION

ACTION Signals:
tonGoingUp(IN:= eRunningState	=	E_LidFeederState.eGoingUp, PT:=T#1500MS);
END_ACTION

ACTION Statistics:



rtrigCycleTimerRead(CLK:=eRunningState=E_LidFeederState.eLidPutted);
IF rtrigCycleTimerRead.Q THEN
	tCycleTime:=tonCycleTimer.ET;
END_IF
tonCycleTimer(IN:=eRunningState>E_LidFeederState.ePuttingLid,PT:=T#1D);
END_ACTION

END_FUNCTION_BLOCK

// ---- POUs/FB/FB_TempRegulator.TcPOU
(*
Nazwa:			FB_TempRegulator
Opis:			Regulator temepratury
Wersja:			v0.1
Data:			2019-07-02
Autor:			DP
Urzadzenia:		Grzałka, czujnik
Konfiguracja:	
Info: 
*)

FUNCTION_BLOCK FB_TempRegulator
VAR_INPUT
	bEnable:BOOL;				(*Zezwolenie na prace regulatora*)
	bEStop:BOOL;				(*Stop Awaryjny nieaktywny*)
	rSetTemp:REAL;				(*Zadana temperatura*)
	rActualTemp:REAL;			(*Aktualna temperatura*)
	rMaxTemp:REAL;				(*Temperatura maksymalna*)
	nRegulatorType:UINT; 		(*0->Regulator PID1, 1->Regulator PID2, 2->Regulator On/Off*)
	PID_:BOOL;
	rKp:REAL;			 		(*Wzmocnienie proporcjonalne regulatora grzałki*)
	rTd:REAL;			 		(*Czas różniczkowania regulatora grzałki*)
	rTi:REAL;			 		(*Czas całkowania regulatora grzałki*)
	Regulator1_:BOOL;
	rPIDCycleTime:REAL;			(*Interwał regulatora PID*)
	bPIDReset:BOOL;				(*Reset PIDa*)
	bPIDFreeze:BOOL;			(*Zatrzymanie PIDa*)
	rPIDYmin:REAL;				(*Ograniczenie dolne wyjścia*)
	rPIDYmax:REAL;				(*Ograniczenie górne wyjścia*)
	Regulator2:BOOL;
	Regulator3:BOOL;
	bRegulatorOffsetOn:REAL;	(*Offset od temperatury zadanej do włączenia regulatora*)
	bRegulatorOffsetOff:REAL;	(*Offset od temperatury zadanej do wyłączeniaa regulatora*)
END_VAR
VAR_OUTPUT
	bHeating:BOOL;				(*Wyjście grzania*)
	bError:BOOL;
	rPID_OUT:REAL;	
END_VAR
VAR_IN_OUT
	bReset:BOOL;				(*Reset regulatora*)
END_VAR

VAR
	(*Regulator OnOff*)
	bHeatingBasicRegulator:BOOL;

	(*Regulator 1*)
	fbPIDBasic:FB_PIDBasic;
	fbPWMBasic:FB_PWM_BASIC;
	bPIDEnable:		BOOL; 		(*Zezwolenie na załączenie PID*)
	(*Koniec regulator 1*)
	
	(*Regulator 2*)
	bPWM_OUT:BOOL;
	PulseGen: TON;				//Timer wyznaczania pulsów 	
	// Czas tasku
	nDeltaT: LREAL;
	// //Różnica między temperaturą zadaną a aktualną
	lrDeltaTemp: LREAL;
	// Sterowanie PWM przekaźnika grzałki
	nRelayDuty: LREAL;
	// Poprzednia wartość różnicy temperatur zadanej i aktualnej
	lrDeltaTempLast: LREAL;
	// Całka po różnicy temperatury zadanej od aktualnej w czasie nDeltaT
	lrI: LREAL;
	// Liczenie przyrostu
	tonPrzyrost: TON;
	// Ostanio zadana temperatura
	lrLastHeaterTemperatureSV: LREAL;
	rtChange: R_TRIG;
	// Rampa zmiany temperatury
	bChangeTemperatureRamp: BOOL;
	// Wartość rampy zmiany temperatury
	lrTempRamp: LREAL;
	// Przytrzymanie ostatniej wartosci wypełnienia PWM grzałki
	nLatchRelayDuty: LREAL;
	// Początek zmian temperatury
	lrStartTemp: LREAL;
	// Dwie trzecie zadanej temperatury osiągniete
	ft2I3Temp: F_TRIG;
	rtrigCycleTimerRead:R_TRIG;
	(*Koniec regulator 2*)
	
END_VAR

aControl();

ACTION aControl:

(*Zabezpieczenia przed wpisaniem zer*)
IF rKp = 0 THEN rKp:=0.0001; END_IF
IF rTi = 0 THEN rTi:=50000; END_IF
IF rPIDCycleTime <100 THEN rPIDCycleTime:=1000; END_IF


(*Włączenie regulatora*)
IF bEnable AND bEStop THEN
	bPIDEnable := TRUE;
	fbPIDBasic.bReset:=FALSE;
	
	(*Wyjście grzania*)		
	bHeating:=fbPWMBasic.bOut OR bPWM_OUT OR bHeatingBasicRegulator;
	rPID_OUT:=LREAL_TO_REAL(fbPIDBasic.lrY);
	
	(*Zabezpieczenie od temperatury maksymalnej*)
	IF rActualTemp > rMaxTemp THEN
		bHeating := FALSE;
	END_IF
	
	(*Regulator 1, PID_Basic, PWM*)
	IF nRegulatorType = 1 THEN 
		aPIDPWMControl_1();
	(*Regulator 2, PID samorobny*)
	ELSIF nRegulatorType = 2 THEN
		aPIDPWMControl_2();		
	(*Regulator 3, Regulator OnOff*)		
	ELSIF nRegulatorType = 3 THEN		
		aOnOffRegulator_3();
	END_IF
	
ELSE
	bPIDEnable := FALSE;
	fbPIDBasic.bReset:=TRUE;
	bHeating:=FALSE;
END_IF

(*Resetowanie regulatora*)
IF bReset THEN
	fbPIDBasic.bReset:=TRUE;
	bReset:=FALSE;
END_IF
END_ACTION

ACTION aOnOffRegulator_3:
(*Prosty regulator wlacz/wylacz*)
IF rActualTemp<rSetTemp+bRegulatorOffsetOn THEN
	bHeatingBasicRegulator := TRUE;
END_IF
IF rActualTemp>rSetTemp+bRegulatorOffsetOff THEN
	bHeatingBasicRegulator := FALSE;
END_IF
END_ACTION

ACTION aPIDPWMControl_1:
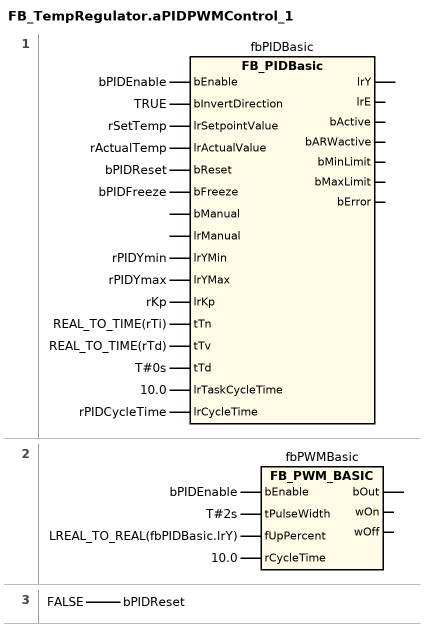
// NETWORK 1
fbPIDBasic(
    bEnable := bPIDEnable,
    bInvertDirection := TRUE,
    lrSetpointValue := rSetTemp,
    lrActualValue := rActualTemp,
    bReset := bPIDReset,
    bFreeze := bPIDFreeze,
    lrYMin := rPIDYmin,
    lrYMax := rPIDYmax,
    lrKp := rKp,
    tTn := REAL_TO_TIME(rTi),
    tTv := REAL_TO_TIME(rTd),
    tTd := T#0s,
    lrTaskCycleTime := 10.0,
    lrCycleTime := rPIDCycleTime); // FB_PIDBasic

// NETWORK 2
fbPWMBasic(
    bEnable := bPIDEnable,
    tPulseWidth := T#2s,
    fUpPercent := LREAL_TO_REAL(fbPIDBasic.lrY),
    rCycleTime := 10.0); // FB_PWM_BASIC

// NETWORK 3
bPIDReset := FALSE;
END_ACTION

ACTION aPIDPWMControl_2:

PulseGen(IN:=bEnable AND NOT PulseGen.Q,PT:=T#1S);
tonPrzyrost(IN:=(bChangeTemperatureRamp AND NOT tonPrzyrost.Q),PT:=T#1S);
ft2I3Temp(CLK:=bChangeTemperatureRamp AND ABS(rSetTemp-rActualTemp)>(ABS(rSetTemp-lrStartTemp)/5),Q=>);
rtChange(CLK:=lrLastHeaterTemperatureSV<>rSetTemp AND bEnable,Q=>);

IF bEnable THEN
	
	//Sterowanie rampą zmiany temperatury zadanej
	IF rtChange.Q OR bChangeTemperatureRamp THEN
		bChangeTemperatureRamp:=TRUE;
		IF rtChange.Q THEN
			lrStartTemp:=rActualTemp;
			lrTempRamp:=rSetTemp;
		END_IF
		
		IF ft2I3Temp.Q THEN
			lrTempRamp:=rActualTemp;
		END_IF
		
		IF rSetTemp>lrTempRamp AND tonPrzyrost.Q AND ABS(rSetTemp-rActualTemp)<(1*ABS(rSetTemp-lrStartTemp)/5) THEN
			lrTempRamp:=lrTempRamp+0.2;
		ELSIF rSetTemp<lrTempRamp AND tonPrzyrost.Q AND ABS(rSetTemp-rActualTemp)<(1*ABS(rSetTemp-lrStartTemp)/5) THEN
			lrTempRamp:=lrTempRamp-0.2;
		END_IF
		
		IF ABS(rSetTemp-lrTempRamp)<=1 AND ABS(rSetTemp-rActualTemp)<(ABS(rSetTemp-lrStartTemp)/5) THEN
			lrTempRamp:=rSetTemp;
			bChangeTemperatureRamp:=FALSE;
		END_IF
		
	END_IF
	
    //REGULATOR PID (regulacja wypełnienia PWM)
	nDeltaT:=UDINT_TO_LREAL(_TaskInfo[1].CycleTime)/10000000;
	lrDeltaTemp:=lrTempRamp-rActualTemp;
		
	lrI:=lrI+((lrDeltaTempLast+lrDeltaTemp)/2)*nDeltaT;
	IF lrI>5000 THEN
		lrI:=5000;
	END_IF
	nRelayDuty:=rKp*(      (*P*)lrDeltaTemp+      (*I*)((1/rTi)*lrI)+     (*D*)(rTd*(lrDeltaTemp-lrDeltaTempLast)/nDeltaT)       );	
	lrDeltaTempLast:=lrDeltaTemp;
	
	IF (rSetTemp-rActualTemp)>0 AND lrI<0 THEN
		lrI:=200;
	END_IF
	
	IF nRelayDuty>1 THEN
		nRelayDuty:=1;
	END_IF
	
	IF nRelayDuty<0 THEN
		nRelayDuty:=0;
	END_IF
	
	IF PulseGen.Q THEN
		nLatchRelayDuty:=nRelayDuty;
	END_IF;	
	bPWM_OUT:=((TIME_TO_LREAL(PulseGen.ET)/TIME_TO_LREAL(PulseGen.PT))<nLatchRelayDuty) AND bEnable;
	
	lrLastHeaterTemperatureSV:=rSetTemp;
ELSE
	lrDeltaTemp:=rSetTemp-rActualTemp;
	lrDeltaTempLast:=lrDeltaTemp;
	nRelayDuty:=0;
	lrI:=0;
END_IF


IF rActualTemp > rSetTemp + 2 THEN
	bPWM_OUT									:= FALSE;
END_IF
END_ACTION

END_FUNCTION_BLOCK

// ---- POUs/FB/Various/FB_PIDBasic.TcPOU
//==================================================================================================
//					Beckhoff Automation Poland
//							18.11.2016
//		Blok funkcyjny regulatora PID w wersji podstawowej
// 	v1.0 	|| TC v 3.1.4020.28 	|| - pierwsza wersja
//==================================================================================================
FUNCTION_BLOCK FB_PIDBasic
VAR_INPUT
	bEnable				: BOOL; 			// Pozdolenie na dzialanie, FALSE - resetuje zawartosc
	bInvertDirection	: BOOL; 			// TRUE: Heating
	lrSetpointValue		: LREAL; 			// Wartosc zadana
	lrActualValue		: LREAL; 			// Wartosc aktualna
	bReset				: BOOL;				// Restart bloku
	bFreeze				: BOOL;				// Zatrzasniecie wyjscia
	bManual				: BOOL;				// Tryb reczny
	lrManual			: LREAL;			// Wartosc dla trybu recznego
	lrYMin				: LREAL;			// Ograniczenie dolne wyjscia
	lrYMax				: LREAL;			// Ograniczenie gorne wyjscia
	lrKp				: LREAL;			// Wzmocnieie proporcjonalne
	tTn					: TIME; 			// Stala czasowa ocji calkujacej
	tTv					: TIME; 			// Stala czasowa akcji rozniczkujacej
	tTd					: TIME; 			// Stala czasowa akcji rozniczkujacej
	lrTaskCycleTime		: LREAL; 			// Czas tasku w ms
	lrCycleTime			: LREAL; 			// Interwal wywolania obliczen w ms - powinna to byc wielokrotnosc cyklu
END_VAR
VAR_OUTPUT
	lrY					: LREAL; 			// Wyjscie
	lrE					: LREAL; 			// Odchylka regulacji
	bActive				: BOOL; 			// Regulator dziala
	bARWactive			: BOOL; 			// Ochrona calkowania
	bMinLimit			: BOOL; 			// Limit gorny
	bMaxLimit			: BOOL; 			// Limit dolny
	bError				: BOOL; 			// Blad parametru
END_VAR
VAR
	bExecutionCycle		: BOOL;
	bInit				: BOOL;
	bIPartEnabled		: BOOL;
	bDPartEnabled		: BOOL;
	bCtrlDisabled		: BOOL;
	uiCycle				: UINT;
	uiCycleCall			: UINT;
	lrTn				: LREAL;
	lrTv				: LREAL;
	lrTd				: LREAL;
	lre_1				: LREAL;
	lrYP				: LREAL;
	lrYI				: LREAL;
	lrYI_1				: LREAL;
	lrYD				: LREAL;
	lrYD_1				: LREAL;
	lrY_1				: LREAL;
	lrdI				: LREAL;
	lrdD				: LREAL;
	lrcD				: LREAL;
	lrY_Test			: LREAL;
END_VAR

	bError		:= FALSE;
	IF lrTaskCycleTime < 0.001 THEN bError := TRUE; END_IF
	IF lrCycleTime < lrTaskCycleTime THEN bError	:= TRUE; END_IF
	IF lrYMin>=lrYMax THEN bError := TRUE; END_IF
	IF (lrKp<0.0) THEN bError := TRUE; END_IF
	IF bError THEN RETURN; 	END_IF


IF NOT bEnable OR NOT bInit	THEN
	lrY				:= 0.0;
	lrE				:= 0.0;
	lrE_1			:= 0.0;
	lrYP			:= 0.0;
	lrYI			:= 0.0;
	lrYI_1			:= 0.0;
	lrYD			:= 0.0;
	lrYD_1			:= 0.0;
	lrY_Test		:= 0.0;
	bARWactive		:= FALSE;
	bActive			:= FALSE;
	uiCycle			:= 1;
	bInit			:= TRUE;
	IF NOT bEnable THEN RETURN; END_IF
END_IF
(* Flagi i limity *)
bActive	:= TRUE;
bIPartEnabled := tTn > t#0ms; (*Czy jest czlon I?*)
bDPartEnabled := tTv > t#0ms; (*Czy jest czlon D?*)
lrManual := LIMIT(lrYMin, lrManual, lrYMax);	(* Manual musi byc w limitach *)

(*Konwersja czasow*)
lrTn	:= TIME_TO_LREAL(tTn);
lrTv	:= TIME_TO_LREAL(tTv);
lrTd	:= TIME_TO_LREAL(tTd);

(*Wyliczenie co ile cykli jest obliczenie wyjscia*)
uiCycleCall := LREAL_TO_UINT(lrCycleTime/lrTaskCycleTime);

(*Obliczenie wspolczynnikow czlonow I i D*)
IF tTn>t#0ms THEN
	lrdI :=	(lrCycleTime/2.0)/lrTn;
END_IF
lrdD :=	lrTv/(lrTd+(lrCycleTime/2.0));
lrcD :=	(lrTd-(lrCycleTime/2.0))/(lrTd+(lrCycleTime/2.0));

(* Obliczenia w kazdym pierwszym cyklu *)
bExecutionCycle := uiCycle = 1;
(* Iterowanie cykli obliczeniowych, obliczenia tylko w cyklu 1, ale to dalej *)
uiCycle:=uiCycle+1;
IF (uiCycle > uiCycleCall) THEN uiCycle:=1; END_IF;

(* Jak obliczenia nie teraz, to wroc *)
IF NOT bExecutionCycle	THEN
	RETURN;
END_IF

(**********************************Regulator PID**********************************)
(*Przepisanie wartosci z poprzedniego cyklu*)
lrE_1	:= lrE;
lrYI_1	:= lrYI;
lrYD_1	:= lrYD;
lrY_1	:= lrY;

(* Kierunek - wprost czy odwrocony*)
lrE := SEL(bInvertDirection, lrActualValue-lrSetpointValue, -(lrActualValue-lrSetpointValue)); (* bInvertDirection = TRUE --> grzanie *)

(*Blokada regulacji gdy mamy minimum i odchylke mniejsza/rowna 0, lub gdy mamy maks i odchylke wieksza/rowna 0*)
bCtrlDisabled:=(bMinLimit AND (lrE <= 0.0)) OR	(bMaxLimit AND (lrE >= 0.0));

(* Jak manual to resetujemy blokadę*)
IF	bManual	THEN bCtrlDisabled:=FALSE; END_IF

bARWactive:=bCtrlDisabled;

(*+++++++++++++++++++++++++++++*)
(*P-I-D-Obliczenia*)
IF NOT bCtrlDisabled	THEN
	(*Czlon: P*);
	lrYP:=lrKp*lrE;
	(*Czlon: I*)
	IF bIPartEnabled THEN
		lrYI:=lrdI*(lrE+lrE_1)+lrYI_1;
	ELSE
		lrYI		:=0;
		lrYI_1	:=0;
	END_IF
	(*Czlon: D*)
	IF bDPartEnabled 	THEN
		IF (lrTd <= lrCycleTime) THEN
			lrYD:= (lrTv/lrCycleTime) * (lrE-lrE_1);
		ELSE
			lrYD:= (lrcD*lrYD_1)+(lrdD*(lrE-lrE_1));
		END_IF
	ELSE
		lrYD		:=0;
		lrYD_1	:=0;
	END_IF
END_IF

(*Sprawdzenie czy nie przekroczymy limitów - w razie potrzeby obcinamy I i D zeby wyrownac do limitu*)
lrY_Test:=lrYP+lrYI+lrYD;
IF NOT bCtrlDisabled THEN
	IF lrY_Test<lrYMin	THEN
		IF		bIPartEnabled THEN
					lrYI:=lrYMin-lrYP-lrYD;
		ELSIF	bDPartEnabled THEN
					lrYD:=lrYMin-lrYP;
		END_IF
	END_IF
	IF lrY_Test>lrYMax THEN
		IF		bIPartEnabled THEN
					lrYI:=lrYMax-lrYP-lrYD;
		ELSIF	bDPartEnabled THEN
					lrYD:=lrYMax-lrYP;
		END_IF
	END_IF
END_IF

(*Jak odciecie sterowania - wyliczenie nowych czlonow I i D*)
IF bCtrlDisabled	THEN
	IF bMinLimit	THEN
		IF		bIPartEnabled THEN
					lrYI:=lrYMin-lrYP-lrYD;
		ELSIF	bDPartEnabled THEN
					lrYD:=lrYMin-lrYP;
		END_IF
	END_IF

	IF bMaxLimit	THEN
		IF		bIPartEnabled THEN
					lrYI:=lrYMax-lrYP-lrYD;
		ELSIF	bDPartEnabled THEN
					lrYD:=lrYMax-lrYP;
		END_IF
	END_IF
END_IF

(*Wyliczenie wyjscia po limitach*)
lrY_Test:=lrYP+lrYI+lrYD;

(*Tryb reczny wyliczenie - wyliczenie nowych czlonow I i D*)
IF bManual	THEN
	IF		bIPartEnabled THEN
				lrYI:=lrManual-lrYP-lrYD;
	ELSIF	bDPartEnabled THEN
				lrYD:=lrManual-lrYP;
	END_IF
END_IF

(*+++++++++++++++++++++++++++++++++++++++++++++++++*)
(*Obliczenie wyjscia*)
lrY:=lrYP+lrYI+lrYD;

(* Freeze - zatrzasniecie wyjscia*)
IF bFreeze THEN
	lrYI			:= lrYI_1;
	lrYD			:= lrYD_1;
	lrY				:= lrY_1;
END_IF

(*Ograniczenie limitów*)
bMaxLimit	:= lrY>=lrYMax;
bMinLimit	:= lrY<=lrYMin;
lrY := LIMIT(lrYMin, lrY, lrYMax);

IF bReset THEN
	A_Reset();
END_IF

ACTION A_Reset:
	bExecutionCycle		:=FALSE;
	bInit				:=FALSE;
	bIPartEnabled		:=FALSE;
	bDPartEnabled		:=FALSE;
	bCtrlDisabled		:=FALSE;
	uiCycle				:=0;
	uiCycleCall			:=0;
	lrTn				:=0;
	lrTv				:=0;
	lrTd				:=0;
	lre_1				:=0;
	lrYP				:=0;
	lrYI				:=0;
	lrYI_1				:=0;
	lrYD				:=0;
	lrYD_1				:=0;
	lrY_1				:=0;
	lrdI				:=0;
	lrdD				:=0;
	lrcD				:=0;
	lrY_Test			:=0;
	lrY					:=0; (* Wyjscie  *)
	lrE					:=0; (* Odchylka regulacji *)
	bActive				:=FALSE; (* Regulator dziala *)
	bARWactive			:=FALSE; (* Ochrona calkowania *)
	bMinLimit			:=FALSE; (* Limit gorny *)
	bMaxLimit			:=FALSE; (* Limit dolny *)
	bError				:=FALSE; (* Blad parametru *)
END_ACTION

END_FUNCTION_BLOCK

// ---- POUs/FB/NC/FB_PWM_BASIC.TcPOU
(********************************************************************************************************)
(*								Beckhoff Automation Poland												*)
(* 									FB_PWM_BASIC v1.1													*)
(* 										22.04.2010														*)
(*	v 1.1 - dodano bEnable, rCycleTime, początkowa faza to wyjście załączone, końcowa wyłączone			*)
(* 		Blok funkcyjny sterowania wyjsciem bOut typu BOOL na zasadzie modulowania szerokosci impulsu.	*)
(*					 Dokladnosc szerokosci impulsu  do 1 cylku sterownika.								*)
(* 							Konieczne jest dodanie biblioteki TcSystem									*)
(*______________________________________________________________________________________________________*)
FUNCTION_BLOCK FB_PWM_BASIC
VAR_INPUT
	bEnable: 			BOOL	:=TRUE;	(* Pozwolenie na działanie bloczka *)
	tPulseWidth: 		TIME; 			(*Szerokosc impulsu = 100% w ms typ zmiennej TIME*)
	fUpPercent: 		REAL; 			(*Aktualne procentowe wypelnienie impulsu*)
	rCycleTime: 		REAL;			(* Czas cylku - task, w milisekundach *)
END_VAR
VAR_OUTPUT
	bOut: 				BOOL;			(* Wyjscie *)
	wOn: 				WORD;			(* Liczba cykli z załączonym wyjściem *)
	wOff: 				WORD;			(* Liczba cykli z wyłaczonym wyjściem *)
END_VAR
VAR
	fCyclePulseWidth: 	REAL;  			(*Dlugosc impulsu = 100% w cyklach typ zmiennej REAL *)
	fCyclesOn: 			REAL;			(*Ilosc cykli, w ktorych sygnal jest zalaczony*)
	State: 				BYTE:=1;		(*Zmienna wyboru w instrukcji CASE*)
	(*Przeliczenie na pelne cykle*)
	wWidth: 			WORD;
	wCycleCounter:		WORD;			(*Licznik cykli zalaczenia/wylaczenia*)
	(*Przechowanie wartosci do porownania*)
	tPulseWidthOld: 	TIME	:= T#0MS;
	fUpPercentOld: 		REAL	:= -1;
END_VAR

IF bEnable THEN
	(*Przelicz tylko gdy zmienia sie dane*)
	IF tPulseWidth <> tPulseWidthOld OR fUpPercent <> fUpPercentOld THEN
		(*Sprawdzamy poprawnosc wprowadzonych danych*)
		IF fUpPercent <0 THEN fUpPercent := 0; END_IF
		IF fUpPercent > 100 THEN fUpPercent := 100; END_IF
		(*Obliczamy*)
		fCyclePulseWidth := TIME_TO_REAL(tPulseWidth)/rCycleTime; (*Dlugosc impulsu*)
		fCyclesOn := fCyclePulseWidth * fUpPercent/100;(*Cykle zalaczenia*)
	
		(*Przeliczamy na pelne cykle*)
		(*Opcja dla dokladniejszego przyblizenia impulsu On i Off*)
		wWidth := REAL_TO_WORD(fCyclePulseWidth);
		wOn := REAL_TO_WORD(fCyclesOn);
		(* Jeśli nie ma takiej potrzeby, nie wystawiaj wyjscia *)
		IF wOff = 0 THEN State := 0; END_IF
		wOff := REAL_TO_WORD(fCyclePulseWidth - fCyclesOn);
		(*Podstawiamy*)
		tPulseWidthOld := tPulseWidth;
		fUpPercentOld := fUpPercent;
	END_IF

	(*Albo wystawiamy TRUE albo FALSE*)
	CASE State OF
		0:
			bOut := FALSE;									(*Ustaw bOut na FALSE*)
			wCycleCounter := wCycleCounter  +  1;			(*Dodaj cykl do licznika*)
			IF wCycleCounter >= wOff THEN					(*Jezeli bylo bOut = FALSE wystarczajaca ilosc cykli to...*)
				wCycleCounter := 0;							(*Resetuj licznik*)
				IF wOff <> wWidth THEN State := 1; END_IF 	(*Przelacz tylko jesli ma byc kiedys bOut = TRUE*)
			END_IF
		1:
			bOut := TRUE;									(*Ustaw bOut na TRUE*)
			wCycleCounter := wCycleCounter  +  1;			(*Dodaj cykl do licznika*)
			IF wCycleCounter >= wOn THEN					(*Jezeli bylo bOut = TRUE wystarczajaca ilosc cykli to...*)
				wCycleCounter := 0;							(*Resetuj licznik*)
				IF wOn <> wWidth THEN State := 0; END_IF 	(*Przelacz tylko jesli ma byc kiedys bOut = FALSE*)
			END_IF
	END_CASE
ELSE
	bOut := FALSE;
	wCycleCounter := 0;
	State := 1;
END_IF

END_FUNCTION_BLOCK

// ---- POUs/FB/FB_JiesangActuatorEncoder_1.TcPOU
(*
Nazwa:			FB_JiesangActuatorEncoder
Opis:			Obsługa podnosnika Jiesang
Wersja:			v0.1
Data:			2018-10-10
Autor:			TW
Urzadzenia:		waga HBM
Konfiguracja:	
Info: 
- podlaczenie po RS485
*)

///!!!!!WAŻNE!!!!!!!!!!
///ABY ENKODER PRACOWAŁ POPRAWNIE TASK PLC MUSI BYĆ USTAWIONY NA 3ms!!!!!!!!!
///Wynika to z faktu że korzystamy ze zwykłych wejść cyfrowych a nie szybkich liczników!!!


FUNCTION_BLOCK FB_JiesangActuatorEncoder_1
VAR_INPUT
	bUpDirectionOut:BOOL;  	//Zmienna sterownika bezpośrednio sterująca siłownikiem w górę (zlinkowana z wyjściem sterownika)
	bDownDirectionOut:BOOL;	//Zmienna sterownika bezpośrednio sterująca siłownikiem w dół (zlinkowana z wyjsciem sterownika)
	bEncoderPulse:BOOL;		//Sygnał impulsów enkodera siłownika
	bHomingCancel:BOOL;		//Anulowanie bazowania enkodera
	bPositionSet:BOOL;		//Zmienna ustawia aktualną wartości pozycji zawartą w zmiennej 'nPositionOffset'
	rPositionOffset:REAL;		//Wartość do nadpisania aktualnej pozycji po ustawieniu wejścia 'AcbtorPositionSet'
	rPulseRatioUp:REAL;			//Przelicznik impulsów na mm  (pokonana_odleglosc_w_mm/ilość_impulsów)
	rPulseRatioDown:REAL;		//Przelicznik impulsów na mm  (pokonana_odleglosc_w_mm/ilość_impulsów)
END_VAR
VAR_OUTPUT
	bHomingDone:BOOL;
	lrActuatorPosition:LREAL:=-200;
	lrPulseRised:LREAL;
	lrPulseFalled:LREAL;
END_VAR
VAR
rtEncoderPulse:R_TRIG;  //wykrywanie zbocza narastającego impulsu encodera
ftEncoderPulse:F_TRIG;  //wykrywanie zbocza opadającego impulsu encodera
rtActuatorPositionSet:R_TRIG;
bLastDirectionUp:BOOL;
rtHomingCancel: R_TRIG;
lrEncoderPulses:LREAL;
END_VAR



//Kasowanie pozycjonowania enkodera
rtHomingCancel(CLK:=bHomingCancel,Q=>);
IF rtHomingCancel.Q THEN
	bHomingDone:=FALSE;
	lrActuatorPosition:=-200;
END_IF

//Jeśli na wejsciu pojawi sie ustawianie aktualnej pozycji enkodera
rtActuatorPositionSet(CLK:=bPositionSet,Q=>);
IF rtActuatorPositionSet.Q THEN
	lrActuatorPosition:=rPositionOffset;
	bHomingDone:=TRUE;
	lrPulseRised:=0;
	lrPulseFalled:=0;
END_IF


//Zapisywanie ostatniego kierunku ruchu siłownika
IF bUpDirectionOut AND NOT bDownDirectionOut THEN
	bLastDirectionUp:=TRUE;
ELSIF bDownDirectionOut AND NOT bUpDirectionOut THEN
	bLastDirectionUp:=FALSE;	
END_IF

//Wykrywanie zbocza pulsu enkodera
rtEncoderPulse(CLK:=bEncoderPulse,Q=>);
ftEncoderPulse(CLK:=bEncoderPulse,Q=>);

IF rtEncoderPulse.Q OR ftEncoderPulse.Q THEN
	lrEncoderPulses	:=	lrEncoderPulses + 1;
	IF bLastDirectionUp THEN
		lrActuatorPosition:=lrActuatorPosition+rPulseRatioUp;
	ELSE
		lrActuatorPosition:=lrActuatorPosition-rPulseRatioDown;
	END_IF
END_IF;

END_FUNCTION_BLOCK

// ---- POUs/FB/NewFBs/FB_Gate.TcPOU
(*
Nazwa:		FB_Gate
Opis:		Szlaban, siłownik
Wersja:		V0.1
Data:		22.05.2024
Autor:		DP
Urządzenia:	Jeden siłownik
Ostatnie zmiany:
	- RRRR-MM-DD [KTO?] Tekst Tekst Tekst Tekst Tekst Tekst Tekst Tekst Tekst Tekst 

Konfiguracja:
	- Krokówka
	Instukcja:
		-
		-
		-
	
Info:
	- Obsługa tylko jednego siłownika

*)

FUNCTION_BLOCK FB_Gate
VAR_INPUT
	bEnable										: BOOL;				//Zezwolenie na pracę
	bEStop										: BOOL;				//Stop awaryjny włączony
	bRun										: BOOL;				//Rozkaz przeciagania
	bHoming										: BOOL;				//Zezwolenie na wykonanie bazowania i pozycjonowanie układu
	bHeightSet									: BOOL;				//Ustaw do pozycji
	bIgnoreError								: BOOL;				//Ignorowanie błędów 
	bReset										: BOOL;				//Reset błędu, jeśli jest w stanie "eError"
	bResetCycle									: BOOL;				//Reset cyklu
	bUpSensor									: BOOL;				//
	bDownSensor									: BOOL;				//
	
	bManualMovement								: BOOL;				//Zezwolenie na ruchy ręczne

	_ALARMINFO_									: BOOL;
	iStationIndex								: UDINT;
	sStationName								: WSTRING;
END_VAR

VAR_OUTPUT
	eState										: E_Station;
	eRunningState								: E_Barrier;			// Stan 
	bError										: BOOL;					// Błąd stacji
	udiErrorID									: UDINT;				// Nr blędu 
	sErrorDescription							: STRING(200);			// Opis błędu
	sErrorDescription2							: STRING(200);			// Opis błędu
	sErrorStationName							: STRING;				// Nazwa stacji
	udiStationID								: UDINT;				// Nr stacji

	bActuator									: BOOL;					
				
	
	bCycleDone									: BOOL;					//Sygnał zakończenia cyklu
	bCycleNotDone								: BOOL;
	bHomingDone									: BOOL;
	tCycleTime									: TIME;					//Czas cyklu
	//Dodatkowe	
	eRunningStateBeforeEStop					: E_Barrier;			//Stan przed E-Stopem	
	bWasErrorOrEstop							: BOOL;
	
END_VAR

VAR
	(*LastStates*)
	eLastState									: E_Station;						//Stan ogólny bloku
	eLastStateTemp								: E_Station;						//Stan ogólny bloku
	eLastRunningState							: E_Barrier;						//Stan podbloku
	eLastRunningStateTemp						: E_Barrier;						//Stan podbloku
	            		
	(*Control*)
	tonResetting								: TON;								//Czas resetu
	tonHoming									: TON;
	tonPreparingToReady							: TON;								//Czas potrzeby na przygotowanie osi
	rtResetCommands								: R_TRIG;                                    	
	rtResetCycle								: R_TRIG;
	tonEstopDelay								: TON;
	
	(*Statistics*)
	tonCycleTimer								: TON;								//Czas cyklu przeciągania	
	rtrigCycleTimerRead							: R_TRIG;

	(*Homing*)
	iHomingCase									: INT;
	
	(*Aborting*)
	iAbortingCase								: INT;
	                                    	
	(*Errors*)
	bStateError									: BOOL;
	bResetCycleOn								: BOOL;
	tonUpSensor									: TON;	
	tonDownSensor								: TON;		
	
	(*Running*)

	tonNotDragActuatorDelay						: TON;
	tonRunningDraging							: TON;
	
	(*Inne*)
	
	iTest: INT;
	iTest1: INT;
	
		//Zmienne od EVENTLOGGER
	bAlarmInit 						: BOOL := TRUE; 
	nAlarmNumerator					: INT;
	arfbAlarm						: ARRAY[0..19] OF  FB_TcAlarm;		//Tablica bloczków błędów
	fbSourceInfo 					: FB_TcSourceInfo;
	iSourceInfo						: I_TcSourceInfo;
	sAlarmTest						: STRING;
	//Koniec zmiennych od EVENTLOGGER
	
END_VAR
	
VAR_IN_OUT
	bManualActuator								: BOOL;		

END_VAR

Signals();
ResetAll();
ErrorHandling();
Control();
Limits();
Statistics();
aStationID();

(*Zapisywanie ostatniego stanu*)
IF eLastStateTemp<>eState THEN
	eLastState := eLastStateTemp;
END_IF
eLastStateTemp := eState;
IF eLastRunningStateTemp<>eRunningState THEN
	eLastRunningState := eLastRunningStateTemp;
END_IF
eLastRunningStateTemp := eRunningState;
(*Koniec Zapisywanie ostatniego stanu*)

ACTION aStationID:
udiStationID	:=	iStationIndex;
END_ACTION

ACTION Control:
	(*****Wyłączenie enable*****)
	IF NOT bEnable AND NOT bError THEN
		IF eState <> E_Station.eDisabled AND eState <> E_Station.ePreparingToDisable THEN
				eState 								:= E_Station.ePreparingToDisable; 
		END_IF	
	END_IF

	(*****Estop*****)
	IF NOT bEstop  THEN	
		IF eState <> E_Station.eAborted AND eState <> E_Station.eAborting AND eState <> E_Station.eDisabled THEN
				eRunningStateBeforeEStop			:= eRunningState;
				eState 								:= E_Station.eAborting; 
				iAbortingCase						:= 0; 
		END_IF
	END_IF


	
CASE eState OF
	
//==========================================================================================	
	E_Station.eDisabled: 						// Stan nieaktywnosci (Stacja wyłączona) 
		
		IF bEnable THEN
			eState 									:= E_Station.ePreparingToReady; 
		END_IF 

//==========================================================================================	    
	E_Station.eAborted: 						// Stan bezpiecznego zatrzymania (po Abortingu) 	
			
		IF bEStop THEN
			bWasErrorOrEstop						:= TRUE;	
			eState 									:= E_Station.ePreparingToReady;
		END_IF		
			
//==========================================================================================	
	E_Station.eAborting:                 		// Stan bezpiecznego zatrzymywania (po EStopie)
		
		CASE iAbortingCase OF
			
			0: //Inicjalizacja
				iAbortingCase						:= 10;
				                                	
			10: //                              	
				iAbortingCase						:= 20;
		                                        	
			20: //Kasowanie komend              	
				//ResetCommands();                					                                                  	
				bManualActuator						:=	FALSE;		                                                      																			
				bResetCycleOn						:=	FALSE;					
				iHomingCase							:=	0;														
 				iAbortingCase						:=	40;
                                               	
			30: //Wyłączenie osi                	
				iAbortingCase						:= 30;
				                                	
			40: //Kasowanie podzespołow         	
				ResetCommands();                	
				iAbortingCase						:= 50;
				                                	
			50: //Przejście do Aborted          	
				iAbortingCase						:= 0;
				eState								:= E_Station.eAborted;
				eRunningState						:= E_Barrier.eReady;
				
		END_CASE

//==========================================================================================			
	E_Station.eError:                 	 		// Stan błędu 	
		
		bWasErrorOrEstop							:= TRUE;

		IF bReset THEN
			eState									:= E_Station.eResetting;	
		ELSE
			ResetCommands();
		END_IF
			
//==========================================================================================
	E_Station.eResetting:						// Stan resetowania bledu (po Errorze)
			
	//Procedura obsługi resetu w zależności od błędu
//	CASE (udiErrorID - iStationIndex) OF 
	bActuator							:= FALSE;		
// 	CASE udiErrorID OF 
// 
// 		131://Error 1 - Błąd siłownika przeciągania
// 			bActuator							:= FALSE;			
// 			bError								:= FALSE;	
// 			iTest :=	iTest	+	1;
// 		132://Error 2 - Błąd siłownika przeciągania
// 			bActuator							:= FALSE;			
// 			bError								:= FALSE;		
// 	
// 	END_CASE
	iTest1 :=	iTest1	+	1;
	
	IF NOT bError THEN
		udiErrorID									:= 0;
		sErrorDescription							:= '';
		sErrorDescription2							:= '';	
		eState										:= E_Station.ePreparingToReady;
	ELSIF tonResetting.Q THEN                   	
		eState										:= E_Station.eError;
	END_IF	
 
//==========================================================================================
	E_Station.eManualMovement:     				// Stan ruchów manualnych  
       
		ManualMovements();
		//Wyjście z trybu serwisowego
		IF NOT bManualMovement THEN
			bActuator								:=	bManualActuator;	
			eState									:=	E_Station.eReady;
		END_IF 

//==========================================================================================		
	E_Station.eHoming:							// Stan bazowania 
		
		Homing();	
		IF NOT bHoming AND NOT bHeightSet AND tonHoming.Q THEN
			eState									:=	E_Station.ePreparingToReady;
		END_IF		
			
//==========================================================================================
	E_Station.eHomingDone:                  	// Stan wykonania bazowania 

		bHomingDone									:= TRUE;
		bResetCycleOn								:= FALSE;		
		IF NOT bHoming AND NOT bHeightSet AND NOT bResetCycleOn THEN
		//	eState									:=	E_Station.eReady;
			eState									:=	E_Station.ePreparingToReady;
		END_IF

//==========================================================================================
	E_Station.ePreparingToReady:            	// Stan przygotowywania do gotowosci (zawsze przed Ready)  

		IF tonPreparingToReady.Q THEN
							
				ResetCommands();
				eState								:= E_Station.eReady;
				eRunningState						:= E_Barrier.eReady;
				
				IF bResetCycleOn THEN
					eState							:= E_Station.eHoming;
				END_IF
				
		END_IF			

//==========================================================================================
	E_Station.ePreparingToDisable:         	 	// Stan przygotowywania do nieaktywnosci (po wyłączeniu Enable) 
		
		bWasErrorOrEstop							:= FALSE;
		bHomingDone									:= FALSE;	
		
		ResetCommands();
		eState										:=	E_Station.eDisabled;
		eRunningState								:=	E_Barrier.eReady;


//==========================================================================================	
	E_Station.eReady:							// Stan gotowosci 


		(*Skasowanie wszystkich komend*)
		IF rtResetCommands.Q THEN	ResetCommands();	END_IF		
	
		IF bRun  (*AND NOT bCycleDone*) THEN
			eState									:= E_Station.eStarting;
		END_IF		
		IF bHoming OR bHeightSet THEN
			eState									:= E_Station.eHoming;
		END_IF
		IF bManualMovement THEN
			bManualActuator							:=	bActuator;							
			eState									:=	E_Station.eManualMovement;					
		END_IF
		IF NOT bRun THEN
			bCycleDone								:= FALSE;
		END_IF

//==========================================================================================
	E_Station.eStopping:					// Stan zatrzymywania 
		
		Running();
		IF eRunningState = E_Barrier.eReady THEN
			eState 									:= E_Station.eReady;
		END_IF


//==========================================================================================
	E_Station.eStarting:                  	// Stan uruchamiania (po Ready)
			
		eState										:= E_Station.eRunning;

//==========================================================================================
	E_Station.eRunning:               		// Stan wykonywania cyklu (po Startingu), w tym stanie osobny
 
		Running();

		IF NOT bRun  THEN					(*Przerywanie cyklu*)
			eState 				 					:= E_Station.eStopping;	
		END_IF
			
		//IF bCycleDone THEN (*Cykl zakończony*)
		//	eState 				 					:= E_Station.eReady;
		//END_IF	
		
//==========================================================================================
END_CASE
END_ACTION

ACTION ErrorHandling:
// Alarm_0200	200	Error	Siłownik | Blokada wysunięcia - sprawdź czujnik lub odblokuj
// Alarm_0201	201	Error	Siłownik | Blokada wsunięcia - sprawdź czujnik lub odblokuj
IF bAlarmInit THEN
    bAlarmInit := FALSE; 
	fbSourceInfo.Clear();
	fbSourceInfo.sName:=wsLiteral_TO_UTF8(sStationName);//'Machine';
	fbSourceInfo.nId:=udiStationID;//2700;
	// Alarm_0200	200	Error	Siłownik | Blokada wysunięcia - sprawdź czujnik lub odblokuj
    arfbAlarm[0].CreateEx(stEventEntry := TC_EVENTS.AlarmClass.Alarm_0200, bWithConfirmation:= FALSE,  ipSourceInfo:= fbSourceInfo); 
	// Alarm_0201	201	Error	Siłownik | Blokada wsunięcia - sprawdź czujnik lub odblokuj
	arfbAlarm[1].CreateEx(stEventEntry := TC_EVENTS.AlarmClass.Alarm_0201, bWithConfirmation:= FALSE,  ipSourceInfo:= fbSourceInfo);
END_IF



//CZYTANIE STATUSÓW
tonEstopDelay			(IN:=bEStop,	PT:=T#3S);
bStateError				:= (eState=E_Station.eError) OR (eState=E_Station.eResetting) OR NOT bEstop OR bIgnoreError;
//bStateError				:= (eState=E_Station.eError) OR (eState=E_Station.eResetting) OR bIgnoreError;

IF bEnable AND tonEstopDelay.Q THEN


	// Alarm_0200	200	Error	Siłownik | Blokada wysunięcia - sprawdź czujnik lub odblokuj
	//Error 1 - Błąd siłownika 
	tonDownSensor	(IN:= bActuator AND NOT bDownSensor	, PT:=T#2S);
	IF tonDownSensor.Q THEN
		IF NOT arfbAlarm[0].bActive THEN
			arfbAlarm[0].Raise(nTimeStamp:=0);
		END_IF
	ELSE	
		IF  arfbAlarm[0].bActive AND bReset THEN
			arfbAlarm[0].Clear(nTimeStamp:=0, bResetConfirmation:= FALSE);
		END_IF	
// 		bError								:= TRUE;
// 		udiErrorID							:= 131;	
// 		//udiErrorID 							:= udiErrorID + iStationIndex;
// 		sErrorDescription					:= 'Siłownik';
// 		sErrorDescription2					:= 'Blokada wysunięcia - sprawdź czujnik lub odblokuj';
	END_IF
	// Alarm_0201	201	Error	Siłownik | Blokada wsunięcia - sprawdź czujnik lub odblokuj
	//Error 2 - Błąd siłownika
	tonUpSensor	(IN:= NOT bActuator AND NOT bUpSensor	, PT:=T#2S);
	IF tonUpSensor.Q THEN
		IF NOT arfbAlarm[1].bActive THEN
			arfbAlarm[1].Raise(nTimeStamp:=0);
		END_IF
	ELSE	
		IF  arfbAlarm[1].bActive AND bReset THEN
			arfbAlarm[1].Clear(nTimeStamp:=0, bResetConfirmation:= FALSE);
		END_IF	

	END_IF;			
		
ELSE
	bError := FALSE;
END_IF

//******************PRZEJŚCIE DO eERROR*****************************

IF bError AND  NOT bStateError THEN
	eState 									:= E_Station.eError;
END_IF

//****************WYŚWIETLANIE STATUSU BLEDU************************
(*Wyświetlanie błedu na wyjściu*)
bError							:= FALSE;
FOR nAlarmNumerator := 0 TO 19 DO
	bError						:= bError OR arfbAlarm[nAlarmNumerator].bActive;
END_FOR

(*Przepisywanie nazwy stacji*)
sErrorStationName 							:= WSTRING_TO_STRING(sStationName);
END_ACTION

ACTION Homing:


IF bHoming THEN // Bazowanie - podjazd do góry i ustawienie obrotu
	CASE iHomingCase OF
	
	0: //
		bHomingDone										:= FALSE;		                                        		
		bActuator										:= FALSE;			
		iHomingCase										:= 10;
	
	10: //
		iHomingCase										:= 20;

	20: //
		iHomingCase										:= 30;
		
	30: //k
		iHomingCase										:= 40;
		
	40: //
		iHomingCase										:= 50;
	
	50: 
		iHomingCase										:= 60;
		
	60: //
		iHomingCase										:= 70;
			
	70:                             	
		iHomingCase										:= 80;

	80:
		iHomingCase										:= 100;
		
	100: //
		iHomingCase										:= 0;
		eState											:= E_Station.eHomingDone;
	
	END_CASE
END_IF	
IF bHeightSet THEN
	bActuator									:= FALSE;	
	eState										:= E_Station.eHomingDone;
END_IF
END_ACTION

ACTION Limits:
(*Wywowyłanie na początku*)


(*Prędkość zakręcania*)


(*Inny parametr*)
//...
END_ACTION

ACTION ManualMovements:

IF NOT bRun AND bManualMovement THEN                        	                                  	                                   	
	bActuator										:=	bManualActuator;			

ELSE
	bManualActuator									:=	FALSE;		
END_IF
	
IF bHoming THEN	
	eState											:=	E_Station.eHoming;	
END_IF                                                	
                                                      	
Running();

IF NOT bRun  THEN
	bCycleDone 										:= FALSE;
	bCycleNotDone 									:= FALSE;	
END_IF
END_ACTION

ACTION ResetAll:
(*****Reset bloczka*****)
IF bEnable THEN
	IF eState <> E_Station.eDisabled AND eState <> E_Station.ePreparingToDisable THEN
		IF bResetCycle THEN
			bResetCycleOn						:= TRUE;
			eState								:= E_Station.ePreparingToReady;
		END_IF
	END_IF
END_IF


IF bResetCycleOn THEN
	
	ResetCommands();
	eRunningState							:= E_Barrier.eReady;	
	eState 				 					:= E_Station.eReady;

END_IF
END_ACTION

ACTION ResetCommands:
//KAsowanie komend ruchu 
                                                     	
bManualActuator											:=	FALSE;		                                                      	
bActuator												:=	FALSE;	
                                                    	
bResetCycleOn											:=	FALSE;	

iHomingCase												:=	0;
//bCycleDone								   				:=	FALSE;
END_ACTION

ACTION Running:
	
CASE eRunningState OF
	
	E_Barrier.eDisabled:
		eRunningState								:= E_Barrier.eReady; 
	
	E_Barrier.eReady:

		//IF NOT bCycleDone  THEN                                           	
			IF bRun THEN   
				bActuator								:=	FALSE;
				eRunningState							:=	E_Barrier.eWaitingToOpen; 
       		END_IF
		//END_IF
		
	E_Barrier.eWaitingToOpen:
	
		bActuator										:=	TRUE;
		IF bDownSensor THEN
			eRunningState								:=	E_Barrier.eOpen; 
		END_IF
	
	E_Barrier.eOpen:	
		bCycleDone										:= TRUE;	
		eRunningState									:= E_Barrier.eDone;	
	
	E_Barrier.eDone:			
		
		IF NOT bRun THEN
			eRunningState								:=	E_Barrier.eWaitingToClose; 
		END_IF
		
	E_Barrier.eWaitingToClose:
	
		bActuator										:=	FALSE;
		IF bUpSensor THEN
			eRunningState								:=	E_Barrier.eReady; 
		END_IF
	

		
END_CASE
END_ACTION

ACTION Signals:

tonPreparingToReady		(IN:=	eState = E_Station.ePreparingToReady			,PT:= T#3S);
tonResetting			(IN:=	eState = E_Station.eResetting					,PT:= T#200MS);
tonHoming				(IN:=	eState = E_Station.eHoming						,PT:= T#1S);
rtResetCommands			(CLK:=	eState = E_Station.eReady 						,Q=>);
END_ACTION

ACTION Statistics:
rtrigCycleTimerRead(CLK:=bCycleDone);
IF rtrigCycleTimerRead.Q THEN
	tCycleTime:=tonCycleTimer.ET;
END_IF
tonCycleTimer(IN:= eRunningState>E_Barrier.eReady, PT:=T#1D);
END_ACTION

END_FUNCTION_BLOCK

// ---- POUs/P06_LidSealer.TcPOU
PROGRAM P06_LidSealer
VAR_INPUT

	IbLidSealerDragHomingSensor 					AT %I* 	:BOOL;				// Czujnik bazowania
	IbLidSealerDragLeadBefore1UpSensor 				AT %I* 	:BOOL;
	IbLidSealerDragLeadBefore1DownSensor 			AT %I* 	:BOOL;
	IbLidSealerDragUpSensor 						AT %I* 	:BOOL; 									// Czujnik pozycji siłownika grzałki zadaniczej góra
	IbLidSealerDragDownSensor 						AT %I* 	:BOOL;										// Czujnik pozycji siłownika grzałki zadaniczej dół
	bMovetoEndPositionLidSealer	:BOOL;
END_VAR


VAR
	
	QbLidSealerBlockActuator 						AT %Q*	: BOOL;  									// Blokada 

	//Grzałka zasadnicza 1
	fbLidSealer												: FB_LidSealer;		
	eLidSealerState											: E_Station; 								// Stan pracy 			
	eLidSealerRunningState									: E_LidSealing; 							// Stan pracy 
	fbLidSealerState										: FB_State;
	
	//WEJŚĆIA I WYJŚĆIA SPRZĘTOWE 1		
	IbLidSealerHeightEncoderPulses 					AT %I*	: BOOL;			
	QbLidSealerHeightUpCmd 							AT %Q*	: BOOL; 									// Wyjście sterujące podnośnikiem siłownika grzałki zadaniczej, Silnik w górę
	QbLidSealerHeightDownCmd 						AT %Q*	: BOOL; 									// Wyjście sterujące podnośnikiem siłownika grzałki zadaniczej, Silnik w dół
	QbLidSealerHeaterPWMOut 						AT %Q*	: BOOL; 									// Wyjście sterujące temperaturą grzałki zadaniczej
	QbLidSealerCoolingFan							AT %Q*	: BOOL;  		

	AIbLidSealerHeaterTempCVSensor 					AT %I*	: INT; 										// Wartość aktualnej temperatury grzałki podajnika platynek
	IbLidSealerTempSensorFailure 					AT %I*	: BOOL;  									// Informacja o uszkodzeniu czujnika temperatury grzałki podajnika platynek
	QbLidSealer_SealingActuator								: BOOL; 									// Sterowanie zaworem podajnika platynek na wyspie zaworowej
	
	//Grzałka zasadnicza 2
	fbLidSealer2											: FB_LidSealer;		
	eLidSealer2State										: E_Station; 								// Stan pracy 			
	eLidSealer2RunningState									: E_LidSealing; 							// Stan pracy 
	fbLidSealer2State										: FB_State;
	
	//WEJŚĆIA I WYJŚĆIA SPRZĘTOWE 2
	IbLidSealer2HeightEncoderPulses 				AT %I*	: BOOL;		
	QbLidSealer2HeightUpCmd 						AT %Q*	: BOOL; 									// Wyjście sterujące podnośnikiem siłownika grzałki zadaniczej, Silnik w górę
	QbLidSealer2HeightDownCmd 						AT %Q*	: BOOL; 									// Wyjście sterujące podnośnikiem siłownika grzałki zadaniczej, Silnik w dół
	QbLidSealer2HeaterPWMOut 						AT %Q*	: BOOL; 									// Wyjście sterujące temperaturą grzałki zadaniczej
	QbLidSealer2CoolingFan							AT %Q*	: BOOL;  	
	
	IbLidSealer2UpSensor 							AT %I*	: BOOL; 									// Czujnik pozycji siłownika grzałki zadaniczej góra
	IbLidSealer2DownSensor 							AT %I*	: BOOL;										// Czujnik pozycji siłownika grzałki zadaniczej dół
	AIbLidSealer2HeaterTempCVSensor 				AT %I*	: INT; 										// Wartość aktualnej temperatury grzałki podajnika platynek
	IbLidSealer2TempSensorFailure 					AT %I*	: BOOL;  									// Informacja o uszkodzeniu czujnika temperatury grzałki podajnika platynek
	QbLidSealer2_SealingActuator							: BOOL; 									// Sterowanie zaworem podajnika platynek na wyspie zaworowej
	IbLidSealerUpSensor								AT %I*	: BOOL;  
	TimerLidSealerEnable									: TOF;
	tonLidSealerEnable										: TON;
	rtEnable												: R_TRIG;

	bTemp													: BOOL;
	bTemp1													: BOOL;
	bTemp2													: BOOL;
	
	//PRZECIAGANIE
	eLidSealerDragStation									: E_Station;
	eLidSealerDragRunningStation							: E_DragStationState;
	fbLidSealerDragState									: FB_State;
	fbLidSealerDragStation									: FB_FormsDragStepper;	
	
	tofLidSealerDragStationEnable							: TOF;
	
	//WEJSCIA I WYJSCIA SPRZETOWE
	QbLidSealerDragLeadBefore1Actuator        				: BOOL;				// Siłownikiem prowadzenia przed 1(1 faza)
	QbLidSealerDragLeadBefore2Actuator        				: BOOL;				// Siłownikiem prowadzenia przed 1(1 faza)
	QbLidSealerDragActuator                	  				: BOOL;				// Siłownikiem przeciągania (1 faza)

	IbLidSealerDragLeadBefore2UpSensor 				AT %I*  : BOOL;				// Czujnik
	
	bLidSealersUp											: BOOL;				//Podnoszenie podajników do góry
	
	//dodatkowa obsługa stopera formatek przy dojeździe 
	
	QbLidSealerStoperActuatorOn	:BOOL;	//		bit to wysterowania sygnału stopera
	lrLidSelaerStoperPosition: LREAL;
	rtLidSealerStoperDraging: R_TRIG;
	rtLidSealerStoperEndingOfDraging2	:R_trig;
	rtLidSelaerStoperPackMLStarting: R_TRIG;
	rtLidSealerStoperEndingOfDraging: R_TRIG;
	bLidSealerStoperWaitingForSensor: BOOL;
	bLidSealerStoperActuatorDelay: BOOL;
	tonbLidSealerStoperActuatorDelay: TON;
	tonSealerStoperActuator	:TON;
	
	//ManualStoper
	rtManualMode	: R_TRIG;
	ftManualMode	: F_TRIG;	
	bLidSealerStoperActuatorLastState	:BOOL;
	
	//Inne
	
END_VAR

IF P00_PackML.fbPMLModeManager.eModeStatus = Tc3_PackML.E_PMLUnitMode.ePMLUnitMode_AUTOMATIC THEN
	
	QbLidSealerBlockActuator 	:=	P00_PackML.fbPMLAuto.ePMLState = Tc3_PackML.E_PMLState.ePMLState_EXECUTE OR 
								P00_PackML.fbPMLAuto.ePMLState = Tc3_PackML.E_PMLState.ePMLState_STOPPING OR 
								P00_PackML.fbPMLAuto.ePMLState = Tc3_PackML.E_PMLState.ePMLState_STARTING;
								
ELSIF P00_PackML.fbPMLModeManager.eModeStatus = Tc3_PackML.E_PMLUnitMode.ePMLUnitMode_MANUAL THEN
	
	QbLidSealerBlockActuator	:= fbLidSealer.bBlockActuator OR fbLidSealer2.bBlockActuator;
	
END_IF
QbLidSealerBlockActuator;

//Wentylatory grzałek
QbLidSealerCoolingFan			:= VIS.lrLidSealer1HeaterTempCV > 50;
QbLidSealer2CoolingFan			:= VIS.lrLidSealer2HeaterTempCV > 50;


bLidSealersUp	:= GVL_IO.IbEmergencyStopButton0Pressed OR GVL_IO.IbEmergencyStopButton1Pressed OR GVL_IO.IbEmergencyStopButton2Pressed OR {warning 'PI odkomentować'}
				   GVL_IO.IbEmergencyStopButton3Pressed OR GVL_IO.IbEmergencyStopButton4Pressed OR IbTurnTableEmergencyStopButtonPressed (*OR IbPucksInserterEmergencyStopButton0Pressed*) OR IbPucksInserterEmergencyStopButton1Pressed 
				OR P07_ROPP.IbROPPEmergencyStopButton0Pressed OR P07_ROPP.IbROPPEmergencyStopButton1Pressed 
				AND (QbLidSealer_SealingActuator OR QbLidSealer2_SealingActuator);
aStoper();
ACT_Limits();
ACT_LidSealer();
ACT_LidSealer2();
ACT_LidSealerDragStation();

//GENEROWANIE STANU STACJI DO WIZKI
fbLidSealerState(
	eState 						:= eLidSealerState , 
	bRun 						:= VIS.bLidSealer1Run,	
	eLidSealingRunningState 	:= eLidSealerRunningState , 
	sStateDesc					=> VIS.sLidSealer1State,
	iState 						=> VIS.iLidSealer1State	);	
	
fbLidSealer2State(
	eState 						:= eLidSealer2State , 
	bRun 						:= VIS.bLidSealer2Run,	
	eLidSealingRunningState 	:= eLidSealer2RunningState , 
	sStateDesc 					=> VIS.sLidSealer2State,
	iState 						=> VIS.iLidSealer2State	);	
	
//PRZEPISYWANIE POMIARÓW
VIS.lrLidSealer1HeaterTempCV := INT_TO_LREAL(AIbLidSealerHeaterTempCVSensor)/10.0;
VIS.lrLidSealer2HeaterTempCV := INT_TO_LREAL(AIbLidSealer2HeaterTempCVSensor)/10.0;

//BAZOWANIE - ZMIAN
tonLidSealerEnable	(IN  := fbLidSealer.bEnable,  PT:=T#5S); (*Dodany ton bo Wizka zjebnie wgrywa zmienne, najpierw włacza Enabla a potem dopiero wybiera recepture*)
rtEnable			(CLK := tonLidSealerEnable.Q, Q=>);
IF rtEnable.Q (*AND eMachineState>=E_MachineState.eReady AND eMachineState<>E_MachineState.eHardError*) THEN //<<-- Mają być stany PackML
	VIS.bLidSealerHeightSet 	:= TRUE;
ELSIF fbLidSealer.eState = E_Station.eHomingDone (*OR eMachineState=E_MachineState.eHardError*) THEN //<<-- Mają być stany PackML
 	VIS.bLidSealerHeightSet	:= FALSE;
END_IF

tonLidSealerEnable	(IN  := fbLidSealer.bEnable,  PT := T#5S); (*Dodany ton bo Wizka zjebnie wgrywa zmienne, najpierw włacza Enabla a potem dopiero wybiera recepture*)
rtEnable			(CLK := tonLidSealerEnable.Q, Q=>);
IF rtEnable.Q AND (P00_PackML.fbPMLAuto.ePMLState = Tc3_PackML.E_PMLState.ePMLState_IDLE OR P00_PackML.fbPMLAuto.ePMLState = Tc3_PackML.E_PMLState.ePMLState_EXECUTE) THEN
    VIS.bLidSealerHeightSet := TRUE;
ELSIF (fbLidSealer.eState = E_Station.eHomingDone AND fbLidSealer2.eState = E_Station.eHomingDone) OR (fbLidSealer.eState = E_Station.eError OR fbLidSealer2.eState = E_Station.eError) THEN//GvlVisualization.bErrorOccure THEN
    VIS.bLidSealerHeightSet := FALSE;
END_IF
(*KONIEC BAZOWANIE - ZMIANA*)

//Opoznienie wyłączanie enabla
TimerLidSealerEnable(IN  := GVL.bLidSealerEnable,   PT := T#2S);

//KASOWANIE ROZKAZÓW CYKLI
IF fbLidSealer.bCycleDone AND GVL.bManualMode THEN
	VIS.bLidSealer1Run 	:= FALSE;
END_IF
IF fbLidSealer2.bCycleDone AND GVL.bManualMode THEN
	VIS.bLidSealer2Run 	:= FALSE;
END_IF

//Przeciąganie
tofLidSealerDragStationEnable(IN:= VIS.bLidSealerDragingStationEnableShow, PT:= T#5S);

ACTION ACT_LidSealer:
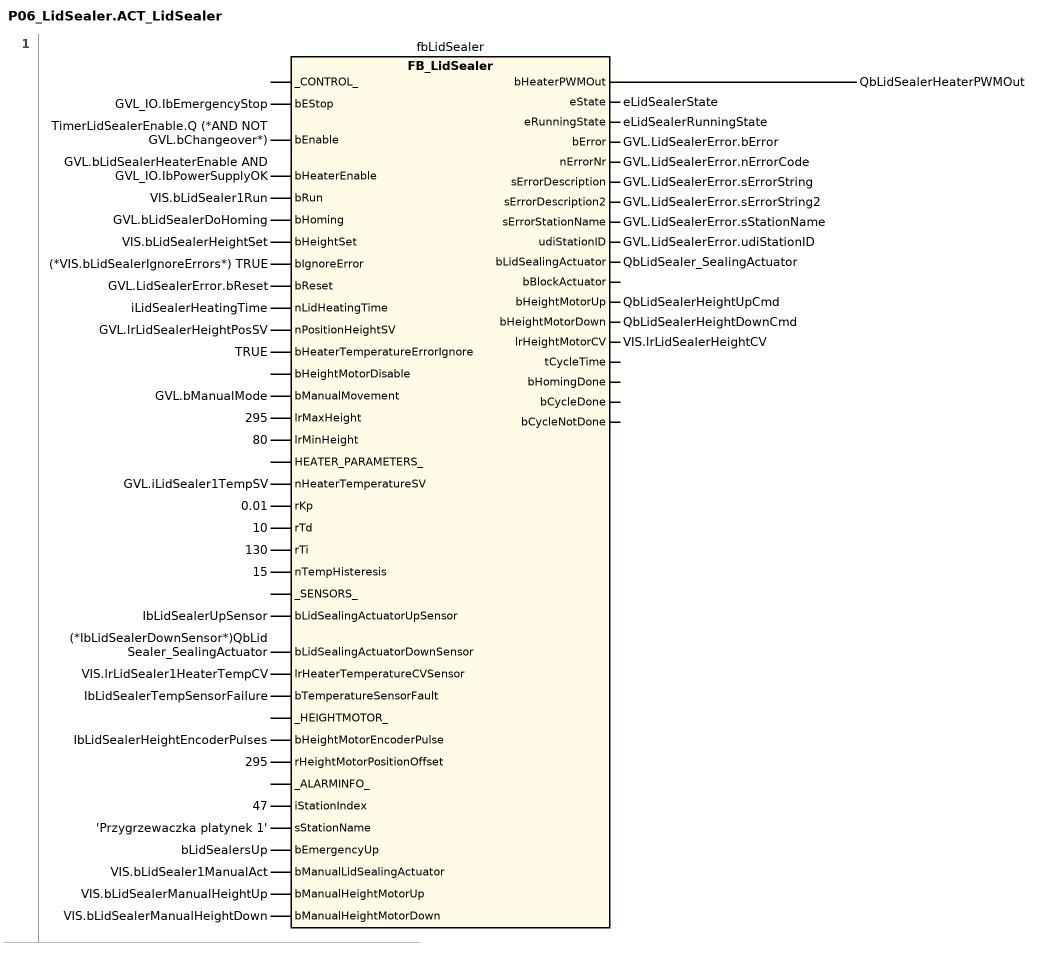
// NETWORK 1
fbLidSealer(
    bEStop := GVL_IO.IbEmergencyStop,
    bEnable := TimerLidSealerEnable.Q (*AND NOT GVL.bChangeover*),
    bHeaterEnable := GVL.bLidSealerHeaterEnable AND GVL_IO.IbPowerSupplyOK,
    bRun := VIS.bLidSealer1Run,
    bHoming := GVL.bLidSealerDoHoming,
    bHeightSet := VIS.bLidSealerHeightSet,
    bIgnoreError := (*VIS.bLidSealerIgnoreErrors*) TRUE,
    bReset := GVL.LidSealerError.bReset,
    nLidHeatingTime := iLidSealerHeatingTime,
    nPositionHeightSV := GVL.lrLidSealerHeightPosSV,
    bHeaterTemperatureErrorIgnore := TRUE,
    bManualMovement := GVL.bManualMode,
    lrMaxHeight := 295,
    lrMinHeight := 80,
    nHeaterTemperatureSV := GVL.iLidSealer1TempSV,
    rKp := 0.01,
    rTd := 10,
    rTi := 130,
    nTempHisteresis := 15,
    bLidSealingActuatorUpSensor := IbLidSealerUpSensor,
    bLidSealingActuatorDownSensor := (*IbLidSealerDownSensor*)QbLidSealer_SealingActuator,
    lrHeaterTemperatureCVSensor := VIS.lrLidSealer1HeaterTempCV,
    bTemperatureSensorFault := IbLidSealerTempSensorFailure,
    bHeightMotorEncoderPulse := IbLidSealerHeightEncoderPulses,
    rHeightMotorPositionOffset := 295,
    iStationIndex := 47,
    sStationName := 'Przygrzewaczka platynek 1',
    bEmergencyUp := bLidSealersUp,
    bManualLidSealingActuator := VIS.bLidSealer1ManualAct,
    bManualHeightMotorUp := VIS.bLidSealerManualHeightUp,
    bManualHeightMotorDown := VIS.bLidSealerManualHeightDown,
    eState => eLidSealerState,
    eRunningState => eLidSealerRunningState,
    bError => GVL.LidSealerError.bError,
    nErrorNr => GVL.LidSealerError.nErrorCode,
    sErrorDescription => GVL.LidSealerError.sErrorString,
    sErrorDescription2 => GVL.LidSealerError.sErrorString2,
    sErrorStationName => GVL.LidSealerError.sStationName,
    udiStationID => GVL.LidSealerError.udiStationID,
    bLidSealingActuator => QbLidSealer_SealingActuator,
    bHeightMotorUp => QbLidSealerHeightUpCmd,
    bHeightMotorDown => QbLidSealerHeightDownCmd,
    lrHeightMotorCV => VIS.lrLidSealerHeightCV); // FB_LidSealer
QbLidSealerHeaterPWMOut := fbLidSealer.bHeaterPWMOut;
END_ACTION

ACTION ACT_LidSealer2:
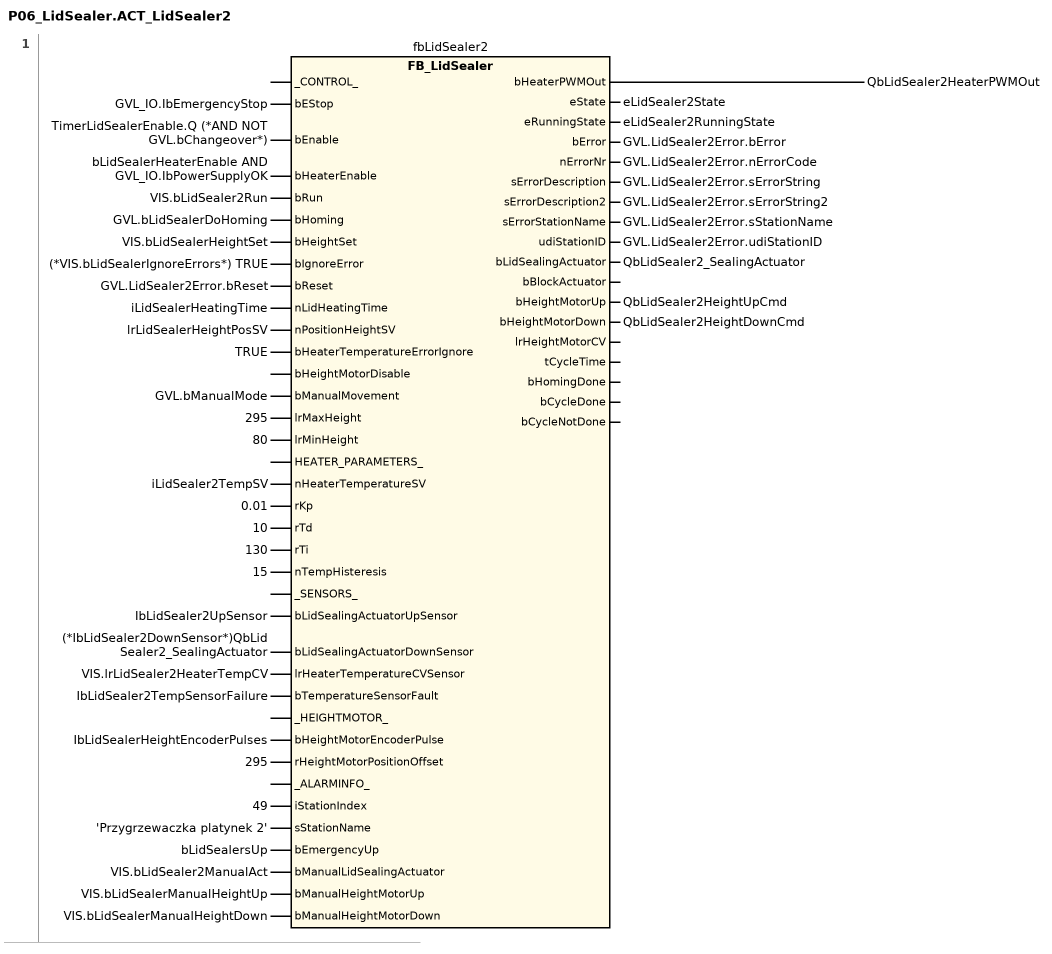
// NETWORK 1
fbLidSealer2(
    bEStop := GVL_IO.IbEmergencyStop,
    bEnable := TimerLidSealerEnable.Q (*AND NOT GVL.bChangeover*),
    bHeaterEnable := bLidSealerHeaterEnable AND GVL_IO.IbPowerSupplyOK,
    bRun := VIS.bLidSealer2Run,
    bHoming := GVL.bLidSealerDoHoming,
    bHeightSet := VIS.bLidSealerHeightSet,
    bIgnoreError := (*VIS.bLidSealerIgnoreErrors*) TRUE,
    bReset := GVL.LidSealer2Error.bReset,
    nLidHeatingTime := iLidSealerHeatingTime,
    nPositionHeightSV := lrLidSealerHeightPosSV,
    bHeaterTemperatureErrorIgnore := TRUE,
    bManualMovement := GVL.bManualMode,
    lrMaxHeight := 295,
    lrMinHeight := 80,
    nHeaterTemperatureSV := iLidSealer2TempSV,
    rKp := 0.01,
    rTd := 10,
    rTi := 130,
    nTempHisteresis := 15,
    bLidSealingActuatorUpSensor := IbLidSealer2UpSensor,
    bLidSealingActuatorDownSensor := (*IbLidSealer2DownSensor*)QbLidSealer2_SealingActuator,
    lrHeaterTemperatureCVSensor := VIS.lrLidSealer2HeaterTempCV,
    bTemperatureSensorFault := IbLidSealer2TempSensorFailure,
    bHeightMotorEncoderPulse := IbLidSealerHeightEncoderPulses,
    rHeightMotorPositionOffset := 295,
    iStationIndex := 49,
    sStationName := 'Przygrzewaczka platynek 2',
    bEmergencyUp := bLidSealersUp,
    bManualLidSealingActuator := VIS.bLidSealer2ManualAct,
    bManualHeightMotorUp := VIS.bLidSealerManualHeightUp,
    bManualHeightMotorDown := VIS.bLidSealerManualHeightDown,
    eState => eLidSealer2State,
    eRunningState => eLidSealer2RunningState,
    bError => GVL.LidSealer2Error.bError,
    nErrorNr => GVL.LidSealer2Error.nErrorCode,
    sErrorDescription => GVL.LidSealer2Error.sErrorString,
    sErrorDescription2 => GVL.LidSealer2Error.sErrorString2,
    sErrorStationName => GVL.LidSealer2Error.sStationName,
    udiStationID => GVL.LidSealer2Error.udiStationID,
    bLidSealingActuator => QbLidSealer2_SealingActuator,
    bHeightMotorUp => QbLidSealer2HeightUpCmd,
    bHeightMotorDown => QbLidSealer2HeightDownCmd); // FB_LidSealer
QbLidSealer2HeaterPWMOut := fbLidSealer2.bHeaterPWMOut;
END_ACTION

ACTION ACT_LidSealerDragStation:
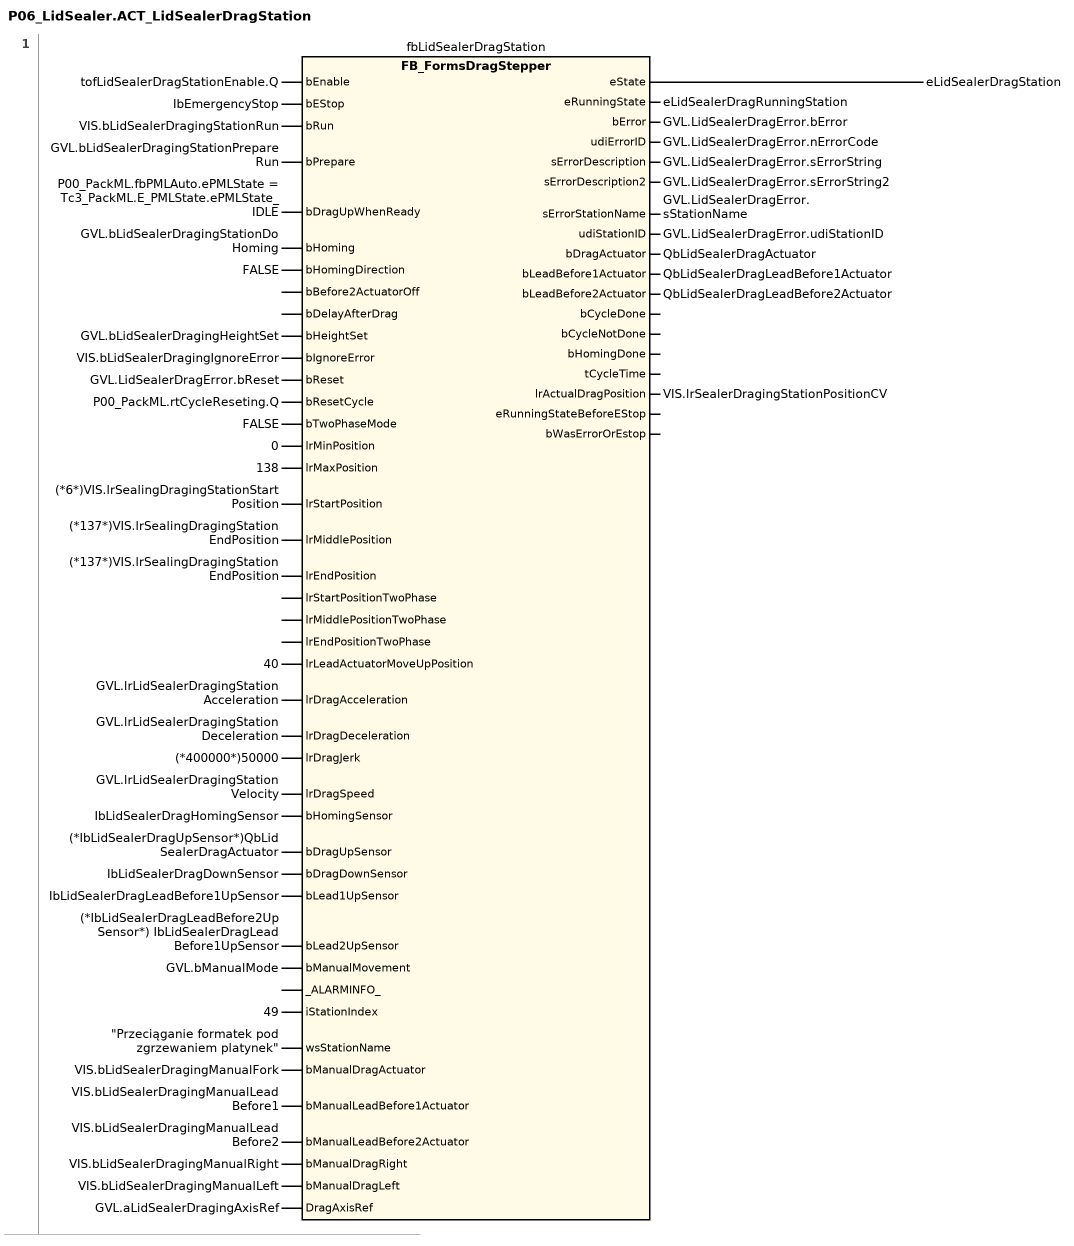
// NETWORK 1
fbLidSealerDragStation(
    bEnable := tofLidSealerDragStationEnable.Q,
    bEStop := IbEmergencyStop,
    bRun := VIS.bLidSealerDragingStationRun,
    bPrepare := GVL.bLidSealerDragingStationPrepareRun,
    bDragUpWhenReady := P00_PackML.fbPMLAuto.ePMLState = Tc3_PackML.E_PMLState.ePMLState_IDLE,
    bHoming := GVL.bLidSealerDragingStationDoHoming,
    bHomingDirection := FALSE,
    bHeightSet := GVL.bLidSealerDragingHeightSet,
    bIgnoreError := VIS.bLidSealerDragingIgnoreError,
    bReset := GVL.LidSealerDragError.bReset,
    bResetCycle := P00_PackML.rtCycleReseting.Q,
    bTwoPhaseMode := FALSE,
    lrMinPosition := 0,
    lrMaxPosition := 138,
    lrStartPosition := (*6*)VIS.lrSealingDragingStationStartPosition,
    lrMiddlePosition := (*137*)VIS.lrSealingDragingStationEndPosition,
    lrEndPosition := (*137*)VIS.lrSealingDragingStationEndPosition,
    lrLeadActuatorMoveUpPosition := 40,
    lrDragAcceleration := GVL.lrLidSealerDragingStationAcceleration,
    lrDragDeceleration := GVL.lrLidSealerDragingStationDeceleration,
    lrDragJerk := (*400000*)50000,
    lrDragSpeed := GVL.lrLidSealerDragingStationVelocity,
    bHomingSensor := IbLidSealerDragHomingSensor,
    bDragUpSensor := (*IbLidSealerDragUpSensor*)QbLidSealerDragActuator,
    bDragDownSensor := IbLidSealerDragDownSensor,
    bLead1UpSensor := IbLidSealerDragLeadBefore1UpSensor,
    bLead2UpSensor := (*IbLidSealerDragLeadBefore2UpSensor*) IbLidSealerDragLeadBefore1UpSensor,
    bManualMovement := GVL.bManualMode,
    iStationIndex := 49,
    wsStationName := "Przeciąganie formatek pod zgrzewaniem platynek",
    bManualDragActuator := VIS.bLidSealerDragingManualFork,
    bManualLeadBefore1Actuator := VIS.bLidSealerDragingManualLeadBefore1,
    bManualLeadBefore2Actuator := VIS.bLidSealerDragingManualLeadBefore2,
    bManualDragRight := VIS.bLidSealerDragingManualRight,
    bManualDragLeft := VIS.bLidSealerDragingManualLeft,
    DragAxisRef := GVL.aLidSealerDragingAxisRef,
    eRunningState => eLidSealerDragRunningStation,
    bError => GVL.LidSealerDragError.bError,
    udiErrorID => GVL.LidSealerDragError.nErrorCode,
    sErrorDescription => GVL.LidSealerDragError.sErrorString,
    sErrorDescription2 => GVL.LidSealerDragError.sErrorString2,
    sErrorStationName => GVL.LidSealerDragError.sStationName,
    udiStationID => GVL.LidSealerDragError.udiStationID,
    bDragActuator => QbLidSealerDragActuator,
    bLeadBefore1Actuator => QbLidSealerDragLeadBefore1Actuator,
    bLeadBefore2Actuator => QbLidSealerDragLeadBefore2Actuator,
    lrActualDragPosition => VIS.lrSealerDragingStationPositionCV); // FB_FormsDragStepper
eLidSealerDragStation := fbLidSealerDragStation.eState;
END_ACTION

ACTION ACT_Limits:
(*
Nazwa:			aSetRecipe
Opis:			Zapisywanie zmiennych gdy mają wartość 0 
Wersja:			v0.1
Data:			2022-06-22
Autor:			DP
Urzadzenia:		
Konfiguracja:	
Info:
- zabezpieczenie przed recepturami które nie mają tych parametrów i jest w nich wartość 0
*)

IF 	VIS.lrSealingDragingStationStartPosition		= 0		THEN	VIS.lrSealingDragingStationStartPosition		:=	5;		END_IF;
IF 	VIS.lrSealingDragingStationEndPosition		= 0		THEN	VIS.lrSealingDragingStationEndPosition		:=	136;	END_IF;
END_ACTION

ACTION aStoper:
								(*
Nazwa:			aStoper
Opis:			Stoper spowalniania formatek
Wersja:			v0.1
Data:			2024-03-21
Autor:			DP
Urzadzenia:		
Konfiguracja:	
Info:

*)
IF NOT vis.bLidFeederEnableShow THEN
	// 0 - Przliczanie od predkości przeciagania				   
	lrLidSelaerStoperPosition	 :=	(188.25 * EXPT(lrBottleDragingStationVelocity,-0.404));
		
	
	// 1 - Wysuwanie stopera na koniec przesuwania gdy pracuje
	rtLidSealerStoperDraging(CLK:=  
									P06_LidSealer.fbLidSealerDragStation.eRunningState = E_DragStationState.eDraging  AND 
									((P00_PackML.fbPMLAuto.ePMLState = E_PMLState.ePMLState_STOPPING) OR  (P00_PackML.fbPMLAuto.ePMLState = E_PMLState.ePMLState_EXECUTE)) AND
							   		P06_LidSealer.fbLidSealerDragStation.lrActualDragPosition > lrLidSelaerStoperPosition+20 
							,Q=>);
							
	IF rtLidSealerStoperDraging.Q THEN
		QbLidSealerStoperActuatorOn	:= TRUE;
	END_IF
	
	
										
	// 2 - Sygnał czekania na czujnik formatek
	rtLidSelaerStoperPackMLStarting (CLK:=  	
												(P00_PackML.fbPMLAuto.ePMLState = E_PMLState.ePMLState_STARTING)
									,Q=>);
	
									
	
	rtLidSealerStoperEndingOfDraging(CLK:=  	P06_LidSealer.fbLidSealerDragStation.eRunningState = E_DragStationState.eDraging AND //P06_LidSealer.fbLidSealerDragStation.eRunningState = E_DragStationState.eDragingDone AND 
												((P00_PackML.fbPMLAuto.ePMLState = E_PMLState.ePMLState_STOPPING) OR  (P00_PackML.fbPMLAuto.ePMLState = E_PMLState.ePMLState_EXECUTE))
									,Q=>);
							
	
	IF rtLidSealerStoperEndingOfDraging.Q OR rtLidSelaerStoperPackMLStarting.Q THEN
		bLidSealerStoperWaitingForSensor	:=	TRUE;	
	END_IF							
	
	// 3 - Wyłączanie stopera
	IF NOT bLidSealerStoperActuatorDelay AND bLidSealerStoperWaitingForSensor AND P00_ReadRFIDCard.bReadedCardLidSealer(*(MAIN.IbLidFeederAfterSensor OR MAIN.IbLidSealerSecondFormSensor)*) THEN
		bLidSealerStoperActuatorDelay	:=	TRUE;
	END_IF
	
	//Zmiana opoznienia dla wolnego transportera
	bFormTransportersDispencerSlowSpeed;
	bDosingTwoPhases;
	IF NOT bFormTransportersDispencerSlowSpeed THEN
			tonbLidSealerStoperActuatorDelay.PT:=T#150MS;//bylo 100
		ELSE
			tonbLidSealerStoperActuatorDelay.PT:=T#650MS; //bylo 500
	END_IF
	
	tonbLidSealerStoperActuatorDelay(IN:=bLidSealerStoperActuatorDelay);
	
	IF tonbLidSealerStoperActuatorDelay.Q THEN
		bLidSealerStoperActuatorDelay		:=	FALSE;
		bLidSealerStoperWaitingForSensor	:=	FALSE;
		QbLidSealerStoperActuatorOn			:=	FALSE;
	END_IF
ELSE
	//rtLidSealerStoperEndingOfDraging2(CLK:=  	P06_LidSealer.fbLidSealerDragStation.eRunningState = E_DragStationState.eDragingDone AND 
	//											((P00_PackML.fbPMLAuto.ePMLState = E_PMLState.ePMLState_STOPPING) OR  (P00_PackML.fbPMLAuto.ePMLState = E_PMLState.ePMLState_EXECUTE))
	//								,Q=>);
	//tonSealerStoperActuator	(IN:= P00_packML.fbIbLidFeederAfterSensor.bOUT AND NOT 
	//		P00_packML.tonLidSealerThirdFormsSensor.q AND NOT P00_packML.tonLidSealerFirstFormsSensor.q AND rtLidSealerStoperEndingOfDraging2.Q, PT:=T#100MS);
	//IF tonSealerStoperActuator.Q THEN
	//	QbLidSealerStoperActuatorOn	:= TRUE;
	//ELSE
	//	QbLidSealerStoperActuatorOn	:= FALSE;	
	//END_IF

	QbLidSealerStoperActuatorOn	:= FALSE;

END_IF
	
	//Manual
	rtManualMode	(CLK:=bManualMode,	Q=>);
	ftManualMode	(CLK:=bManualMode,	Q=>);
	IF rtManualMode.Q THEN
		bLidSealerStoperActuatorLastState	:=	QbLidSealerStoperActuatorOn;
		VIS.bLidSealerStoperManualActuator	:=	QbLidSealerStoperActuatorOn;
	END_IF
	IF bManualMode THEN
		QbLidSealerStoperActuatorOn			:=	VIS.bLidSealerStoperManualActuator;
	END_IF
	IF ftManualMode.Q THEN
		QbLidSealerStoperActuatorOn			:= bLidSealerStoperActuatorLastState;
	END_IF
	// Koniec Manual
END_ACTION

END_PROGRAM

// ---- POUs/FB/FB_LidSealer.TcPOU
(*
Nazwa:			FB_LidSealer
Opis:			Zgrzewarka platynek
Wersja:			v1.0
Data:			2019-07-02
Autor:			TW,DP,MP
Urzadzenia:		Podnosnik stacji, grzałka, silownik
Konfiguracja:	
Info: 
- Dodano błędy od nastaw powyżej max i min (error 7 i 8)
- Dodano do testów inny regulator temperatury
- Zmiana Homingów według CatchStation
*)

FUNCTION_BLOCK FB_LidSealer
VAR_INPUT
	_CONTROL_:BOOL;	
	bEStop:BOOL;						//Stop Awaryjny nieaktywny
	bEnable:BOOL;						//Zezowlenie na pracę grzałki zasadniczej
	bHeaterEnable:BOOL; 				//Zezwolenie na pracę grzałki wstępnej
	bRun:BOOL;
	bHoming:BOOL;						//Zezwolenie na wykonanie bazowania i pozycjonowania podajnika
	bHeightSet:BOOL;					//Ustaw wysokość
	bIgnoreError:BOOL;					//Ignorowania błędów cyklu pracy
	bReset:BOOL;						//Reset błędu, jeśli w stanie "eError"
	nLidHeatingTime:INT;				//Czas zgrzewania wstępnego [ms]
	nPositionHeightSV:LREAL;			//Wysokość zadana na której ma znajdować się podajnik
	bHeaterTemperatureErrorIgnore:BOOL; //Zmienna pozwalająca ignorowanie aktualnej temperatury
	bHeightMotorDisable:BOOL;			//Wyłączenie ruchu podnośnika
	bManualMovement:BOOL; 				//Uruchomienie trybu ruchów ręcznych
	lrMaxHeight:LREAL;					//Maksymalna wysokość grzałki zasadniczej
	lrMinHeight:LREAL;					//Minimalna wysokość grzałki zasadniczej
	HEATER_PARAMETERS_:BOOL;			
	nHeaterTemperatureSV:INT;			//Zadana wartość grzałki grzałki zasadniczej
	rKp:REAL;							//Wzmocnienie proporcjonalne regulatora grzałki
	rTd:REAL;							//Czas różniczkowania regulatora grzałki
	rTi:REAL;							//Czas całkowania regulatora grzałki
	nTempHisteresis:INT;				//Dopuszczalna różnica pomiędzy wartością zadaną a aktualną [st. C]	

	_SENSORS_:BOOL;
	bLidSealingActuatorUpSensor:BOOL;		//krańcówka górna grzałki zasadniczej
	bLidSealingActuatorDownSensor:BOOL;		//krańcówka dolna grzałki zasadniczej
	lrHeaterTemperatureCVSensor:LREAL;		//Wartość aktualna temperatury grzałki
	bTemperatureSensorFault:BOOL;			//Błąd czujnika temperatury
	
	_HEIGHTMOTOR_ :BOOL;	
	bHeightMotorEncoderPulse :BOOL;			//Sygnał impulsów enkodera siłownika
	rHeightMotorPositionOffset :REAL;		//Wysokość bazowani podnośnika

	_ALARMINFO_ :BOOL;
	iStationIndex:UDINT;					//Numer stacji 
	sStationName:STRING;					//Nazwa stacji
	
	bEmergencyUp					: BOOL;
	
END_VAR
VAR_OUTPUT
	bHeaterPWMOut :BOOL;					//Wyjscie PWM sterujące grzałką
	eState: E_Station;						//Stan ogólny bloku
	eRunningState: E_LidSealing;		//Stan podbloku
	bError: BOOL;							//Błąd stacji
	nErrorNr: UDINT;						//Nr błędu grzałki zasadniczej
	sErrorDescription:STRING(200);			//Opis błędu
	sErrorDescription2:STRING(200);			//Opis błędu
	sErrorStationName:STRING;				//Nazwa stacji
	udiStationID:UDINT;						// Nr stacji

	bLidSealingActuator:BOOL;				//Sterownie siłownika Grzałki
	bBlockActuator:BOOL;					//Blokowanie siłownika
	bHeightMotorUp:BOOL;					//Sterowanie silnikiem podnośnika  - RUCH W GÓRĘ
	bHeightMotorDown:BOOL;					//Sterowanie silnikiem podnośnika  - RUCH W DÓŁ
	lrHeightMotorCV:LREAL;					//Aktualna pozycja podnośnika
	tCycleTime:TIME;	
	bHomingDone:BOOL;						//Wymagane ponowne bazowanie (blad podczas bazowania lub stop awaryjny)
	bCycleDone:BOOL;
	bCycleNotDone:BOOL;
END_VAR
VAR

	tonHeatingTime: TON;					//Timer czasu zgrzewania platynki
	tonHeightNoChange: TON; 				//Timer wykrycia braku ruchu siłownika zmiany wysokości stacji
	nLastPositionHeightCV: LREAL;			//Pozycja podnośnika w poprzednim cyklu programu
	tonErrorHeightChange: TON; 				//Timer błędu podnośnika
	tonSealingActuatorUpLag: TON; 			//Timer opóźnienia siłownika zgrzewania po wysterowaniu go w górę
	tonSealingActuatorDownLag: TON; 		//Timer opóźnienia siłownika zgrzewania po wysterowaniu go w dół
	
	rtEncoderHomed:R_TRIG;
	tonCycleTimer:TON;
	rtrigCycleTimerRead:R_TRIG;
	tonLimitPosMinReachedDelay: TON;
	tonLimitPosMaxReachedDelay: TON;

	tonMaxHeight: TON;
	tonMinHeight: TON;
	//Podnośnik Jiesang
	fbHeightMotorEncoder: FB_JiesangActuatorEncoder_1;	// Blok enkodera podnośnika chwytaka stabilizującego pod zakręcarką	
	bHeightMotorEncoderCounterReset:BOOL; 				// Sygnał resetu enkodera
	bHeightMotorEncoderHomed:BOOL;						// Informacja od enkodera że jest zbazowany

	
	eLastState: E_Station;								// Stan ogólny bloku
	eLastRunningState: E_LidSealing;					// Stan podbloku
	eLastStateTemp: E_Station;							// Stan ogólny bloku
	eLastRunningStateTemp: E_LidSealing;				// Stan podbloku

	bStateError: BOOL;

	fbTempRegulator				: FB_TempRegulator;
	bTempRegulatorReset			: BOOL;
	
	tofbHeaterPWMOut					: TOF;
	tonHeaterOnAndNotHeating			: TON;
	lrHeaterTemperatureCVSensorLast		: LREAL;	//Wartość aktualna temperatury grzałki
	tonHeaterOnAndSensorShows0			: TON;

	tonbNOTLidSealingActuator: TON;
	tofHeightMotorDown: TOF;
	tonbBlockActuator: TON;
	rtbHeightMotorEncoderPulse: R_TRIG;
	ftbHeightMotorEncoderPulse: F_TRIG;
	lrHeightMotorEncoderPulses: LREAL;
	
		//Zmienne od EVENTLOGGER
	bAlarmInit 						: BOOL := TRUE; 
	nAlarmNumerator					: INT;
	arfbAlarm						: ARRAY[0..19] OF  FB_TcAlarm;		//Tablica bloczków błędów
	fbSourceInfo 					: FB_TcSourceInfo;
	iSourceInfo						: I_TcSourceInfo;
	sAlarmTest						: STRING;
	//Koniec zmiennych od EVENTLOGGER
END_VAR

VAR_IN_OUT
	bManualLidSealingActuator:BOOL;		//Ruch ręczny siłownika zgrzewającego;
	bManualHeightMotorUp:BOOL;			//Ruch ręczny podnośnika stacji w górę
	bManualHeightMotorDown:BOOL;		//Ruch ręczny podnośnika stacji w dół
END_VAR


HeightMotor();
ErrorHandling();
Control();
HeaterRegulator();
Statistics();
Protections();
EncoderTest();
aStationID();

(*Zapisywanie ostatniego stanu*)
IF eLastStateTemp<>eState THEN
	eLastState := eLastStateTemp;
END_IF
eLastStateTemp := eState;
IF eLastRunningStateTemp<>eRunningState THEN
	eLastRunningState := eLastRunningStateTemp;
END_IF
eLastRunningStateTemp := eRunningState;
(*Koniec Zapisywanie ostatniego stanu*)

nLastPositionHeightCV:=lrHeightMotorCV;

ACTION aStationID:
udiStationID	:=	iStationIndex;
END_ACTION

ACTION Control:
	tofHeightMotorDown(IN:=bHeightMotorDown, PT:=T#1S); //Zabezpieczenie przed zbyt szybkim przełączeniem pomiędzy Down a Up, bezpiecznieki sie palą


	(** TIMERY**)
	rtEncoderHomed(CLK:=bHeightMotorEncoderHomed,Q=>);
	tonHeightNoChange(IN:=((bHeightMotorUp OR bHeightMotorDown) AND (nLastPositionHeightCV=lrHeightMotorCV)), PT:=T#1S); 
	tonLimitPosMinReachedDelay(IN:=(lrHeightMotorCV<=lrMinHeight) AND eState=E_Station.eHoming,PT:=T#2S);
	tonLimitPosMaxReachedDelay(IN:=(lrHeightMotorCV>=lrMaxHeight) AND eState=E_Station.eHoming,PT:=T#2S);
	tonbBlockActuator(IN:=bBlockActuator,PT:=T#1000MS);
	
	(*****Wyłączenie enable*****)
	IF NOT bEnable THEN
		IF eState <> E_Station.eDisabled AND eState <> E_Station.ePreparingToDisable THEN
				eState 				:= E_Station.ePreparingToDisable; 
		END_IF	
	END_IF

